METHOD PUBLIC  Clone : I_Node
VAR
	pNode : POINTER TO Node_F_VN_CopyImageRegionToRegion;
END_VAR
pNode := __NEW(Node_F_VN_CopyImageRegionToRegion);
Clone := pNode^;
END_METHOD

METHOD PROTECTED OnExecute
hresult.Value := F_VN_CopyImageRegionToRegion(
    ipSrcImage := ipSrcImage.Value,
    nXSrc := nXSrc.Value,
    nYSrc := nYSrc.Value,
    nWidth := nWidth.Value,
	nHeight := nHeight.Value,
	ipDestImage := ipDestImage.Value,
    nXDest := nXDest.Value,
    nYDest := nYDest.Value,
	hrPrev:= hrPrev.Value);
END_METHOD

METHOD PUBLIC PreExecutionCheck
VAR_INPUT
	Check : I_PreExecutionChecks;
END_VAR
VAR
    imgWidth : UDINT;
    imgHeight : UDINT;
    roiRectangle : TcVnRectangle_UDINT;
END_VAR
Check.IsTrue(ipSrcImage.IsValid, 'ipSrcImage must contain an image');

IF Check.Failed THEN
    RETURN;
END_IF

ipSrcImage.Value.GetWidth(imgWidth);
ipSrcImage.Value.GetHeight(imgHeight);
roiRectangle.nX := nXSrc.Value;
roiRectangle.nY := nYSrc.Value;
roiRectangle.nWidth := nWidth.Value;
roiRectangle.nHeight := nHeight.Value;

Check.IsTrue(IsRoiSizeOK_Udint(roiRectangle, imgWidth, imgHeight), 'ROI must fit within ipSrcImage');

//TODO Check nXDist and nYDest values?
END_METHOD

END_FUNCTION_BLOCK

// Nodes/Basic Image Ops/Node_F_VN_CopyIntoDisplayableImage
{attribute 'linkalways'} 
{attribute 'no_explicit_call' := 'This FB is a CLASS and must be accessed using methods or properties'}
{attribute 'enable_dynamic_creation'}
FUNCTION_BLOCK Node_F_VN_CopyIntoDisplayableImage EXTENDS VisionNode
VAR
    ipSrcImage : _ITcVnImage;
    ipDestImage : _ITcVnDisplayableImage;
    hrPrev : _HRESULT(S_OK);
	hresult : _HRESULT(S_OK);
END_VAR

METHOD FB_init : BOOL
VAR_INPUT
	bInitRetains : BOOL; // if TRUE, the retain variables are initialized (warm start / cold start)
	bInCopyCode : BOOL;  // if TRUE, the instance afterwards gets moved into the copy code (online change)
END_VAR
AddInput('ipSrcImage', ipSrcImage);
AddInput('hrPrev', hrPrev);
AddOutput('ipDestImage', ipDestImage);
AddOutput('hresult',hresult);
END_METHOD

METHOD PUBLIC  Clone : I_Node
VAR
	pNode : POINTER TO Node_F_VN_CopyIntoDisplayableImage;
END_VAR
pNode := __NEW(Node_F_VN_CopyIntoDisplayableImage);
Clone := pNode^;
END_METHOD

METHOD PROTECTED OnExecute
hresult.Value := F_VN_CopyIntoDisplayableImage(
    ipSrcImage := ipSrcImage.Value,
	ipDestImage := ipDestImage.Value,
	hrPrev:= hrPrev.Value);
END_METHOD

METHOD PUBLIC PreExecutionCheck
VAR_INPUT
	Check : I_PreExecutionChecks;
END_VAR
Check.IsTrue(ipSrcImage.IsValid, 'ipSrcImage must contain an image');
END_METHOD

END_FUNCTION_BLOCK

// Nodes/Basic Image Ops/Node_F_VN_CreateAssociatedImage
{attribute 'linkalways'} 
{attribute 'no_explicit_call' := 'This FB is a CLASS and must be accessed using methods or properties'}
{attribute 'enable_dynamic_creation'}
FUNCTION_BLOCK Node_F_VN_CreateAssociatedImage EXTENDS VisionNode
VAR
    ipSrcImage : _ITcVnImage;
    ipDestImage : _ITcVnImage;
    hrPrev : _HRESULT(S_OK);
	hresult : _HRESULT(S_OK);
END_VAR

METHOD FB_init : BOOL
VAR_INPUT
	bInitRetains : BOOL; // if TRUE, the retain variables are initialized (warm start / cold start)
	bInCopyCode : BOOL;  // if TRUE, the instance afterwards gets moved into the copy code (online change)
END_VAR
AddInput('ipSrcImage', ipSrcImage);
AddInput('hrPrev', hrPrev);
AddOutput('ipDestImage', ipDestImage);
AddOutput('hresult',hresult);
END_METHOD

METHOD PUBLIC  Clone : I_Node
VAR
	pNode : POINTER TO Node_F_VN_CreateAssociatedImage;
END_VAR
pNode := __NEW(Node_F_VN_CreateAssociatedImage);
Clone := pNode^;
END_METHOD

METHOD PROTECTED OnExecute
hresult.Value := F_VN_CreateAssociatedImage(
    ipSrcImage := ipSrcImage.Value,
	ipDestImage := ipDestImage.Value,
	hrPrev:= hrPrev.Value);
END_METHOD

METHOD PUBLIC PreExecutionCheck
VAR_INPUT
	Check : I_PreExecutionChecks;
END_VAR
Check.IsTrue(ipSrcImage.IsValid, 'ipSrcImage must contain an image');
END_METHOD

END_FUNCTION_BLOCK

// Nodes/Basic Image Ops/Node_F_VN_CreateEmptyImage
{attribute 'linkalways'} 
{attribute 'no_explicit_call' := 'This FB is a CLASS and must be accessed using methods or properties'}
{attribute 'enable_dynamic_creation'}
FUNCTION_BLOCK Node_F_VN_CreateEmptyImage EXTENDS VisionNode
VAR
    ipImage : _ITcVnImage;
    hrPrev : _HRESULT(S_OK);
	hresult : _HRESULT(S_OK);
END_VAR

METHOD FB_init : BOOL
VAR_INPUT
	bInitRetains : BOOL; // if TRUE, the retain variables are initialized (warm start / cold start)
	bInCopyCode : BOOL;  // if TRUE, the instance afterwards gets moved into the copy code (online change)
END_VAR
AddInput('hrPrev', hrPrev);
AddOutput('ipImage', ipImage);
AddOutput('hresult',hresult);
END_METHOD

METHOD PUBLIC  Clone : I_Node
VAR
	pNode : POINTER TO Node_F_VN_CreateEmptyImage;
END_VAR
pNode := __NEW(Node_F_VN_CreateEmptyImage);
Clone := pNode^;
END_METHOD

METHOD PROTECTED OnExecute
hresult.Value := F_VN_CreateEmptyImage(
    ipImage := ipImage.Value,
	hrPrev:= hrPrev.Value);
END_METHOD

METHOD PUBLIC PreExecutionCheck
VAR_INPUT
	Check : I_PreExecutionChecks;
END_VAR
END_METHOD

END_FUNCTION_BLOCK

// Nodes/Basic Image Ops/Node_F_VN_CreateImage
{attribute 'linkalways'} 
{attribute 'no_explicit_call' := 'This FB is a CLASS and must be accessed using methods or properties'}
{attribute 'enable_dynamic_creation'}
FUNCTION_BLOCK Node_F_VN_CreateImage EXTENDS VisionNode
VAR
    ipImage : _ITcVnImage;
    nWidth : _UDINT(1);
    nHeight : _UDINT(1);
    ePixelType : _ETcVnElementType(ETcVnElementType.TCVN_ET_USINT);
    nChannelNum : _UDINT(1);
    hrPrev : _HRESULT(S_OK);
	hresult : _HRESULT(S_OK);
END_VAR

METHOD FB_init : BOOL
VAR_INPUT
	bInitRetains : BOOL; // if TRUE, the retain variables are initialized (warm start / cold start)
	bInCopyCode : BOOL;  // if TRUE, the instance afterwards gets moved into the copy code (online change)
END_VAR
AddParameter('nWidth', nWidth);
AddParameter('nHeight', nHeight);
AddParameter('ePixelType', ePixelType);
AddParameter('nChannelNum', nChannelNum);
AddInput('hrPrev', hrPrev);
AddOutput('ipImage', ipImage);
AddOutput('hresult',hresult);
END_METHOD

METHOD PUBLIC  Clone : I_Node
VAR
	pNode : POINTER TO Node_F_VN_CreateImage;
END_VAR
pNode := __NEW(Node_F_VN_CreateImage);
Clone := pNode^;
END_METHOD

METHOD PROTECTED OnExecute
hresult.Value := F_VN_CreateImage(
    ipImage := ipImage.Value,
    nWidth := nWidth.Value,
    nHeight := nHeight.Value,
    ePixelType := ePixelType.Value,
    nChannelNum := nChannelNum.Value,
	hrPrev:= hrPrev.Value);
END_METHOD

METHOD PUBLIC PreExecutionCheck
VAR_INPUT
	Check : I_PreExecutionChecks;
END_VAR
Check.IsTrue((nWidth.Value > 0), 'nWidth must be greater than 0');
Check.IsTrue((nHeight.Value > 0), 'nHeight must be greater than 0');
Check.IsTrue((nChannelNum.Value >= 1), 'nChannelNum must be greater than or equal to 1');
Check.IsTrue((nChannelNum.Value <= 255), 'nChannelNum must be less than or equal to 255');
END_METHOD

END_FUNCTION_BLOCK

// Nodes/Basic Image Ops/Node_F_VN_CreateImageAndSetPixels
{attribute 'linkalways'} 
{attribute 'no_explicit_call' := 'This FB is a CLASS and must be accessed using methods or properties'}
{attribute 'enable_dynamic_creation'}
FUNCTION_BLOCK Node_F_VN_CreateImageAndSetPixels EXTENDS VisionNode
VAR
    ipImage : _ITcVnImage;
    nWidth : _UDINT(1);
    nHeight : _UDINT(1);
    ePixelType : _ETcVnElementType(ETcVnElementType.TCVN_ET_USINT);
    nChannelNum : _UDINT(1);
    aValue : _TcVnVector4_LREAL;
    hrPrev : _HRESULT(S_OK);
	hresult : _HRESULT(S_OK);
END_VAR

METHOD FB_init : BOOL
VAR_INPUT
	bInitRetains : BOOL; // if TRUE, the retain variables are initialized (warm start / cold start)
	bInCopyCode : BOOL;  // if TRUE, the instance afterwards gets moved into the copy code (online change)
END_VAR
AddParameter('nWidth', nWidth);
AddParameter('nHeight', nHeight);
AddParameter('ePixelType', ePixelType);
AddParameter('nChannelNum', nChannelNum);
AddInput('aValue', aValue);
AddInput('hrPrev', hrPrev);
AddOutput('ipImage', ipImage);
AddOutput('hresult',hresult);
END_METHOD

METHOD PUBLIC  Clone : I_Node
VAR
	pNode : POINTER TO Node_F_VN_CreateImageAndSetPixels;
END_VAR
pNode := __NEW(Node_F_VN_CreateImageAndSetPixels);
Clone := pNode^;
END_METHOD

METHOD PROTECTED OnExecute
hresult.Value := F_VN_CreateImageAndSetPixels(
    ipImage := ipImage.Value,
    nWidth := nWidth.Value,
    nHeight := nHeight.Value,
    ePixelType := ePixelType.Value,
    nChannelNum := nChannelNum.Value,
    aValue := aValue.Value,
	hrPrev:= hrPrev.Value);
END_METHOD

METHOD PUBLIC PreExecutionCheck
VAR_INPUT
	Check : I_PreExecutionChecks;
END_VAR
Check.IsTrue((nWidth.Value > 0), 'nWidth must be greater than 0');
Check.IsTrue((nHeight.Value > 0), 'nHeight must be greater than 0');
Check.IsTrue((nChannelNum.Value >= 1), 'nChannelNum must be greater than or equal to 1');
Check.IsTrue((nChannelNum.Value <= 4), 'nChannelNum must be less than or equal to 4');
END_METHOD

END_FUNCTION_BLOCK

// Nodes/Basic Image Ops/Node_F_VN_CreateNDimensionalImage
{attribute 'linkalways'} 
{attribute 'no_explicit_call' := 'This FB is a CLASS and must be accessed using methods or properties'}
{attribute 'enable_dynamic_creation'}
FUNCTION_BLOCK Node_F_VN_CreateNDimensionalImage EXTENDS VisionNode
VAR
    ipImage : _ITcVnImage;
    aShape : _TcVnArray33_UDINT;
    ePixelType : _ETcVnElementType(ETcVnElementType.TCVN_ET_USINT);
    hrPrev : _HRESULT(S_OK);
	hresult : _HRESULT(S_OK);
END_VAR

METHOD FB_init : BOOL
VAR_INPUT
	bInitRetains : BOOL; // if TRUE, the retain variables are initialized (warm start / cold start)
	bInCopyCode : BOOL;  // if TRUE, the instance afterwards gets moved into the copy code (online change)
END_VAR
AddParameter('aShape', aShape);
AddParameter('ePixelType', ePixelType);
AddInput('hrPrev', hrPrev);
AddOutput('ipImage', ipImage);
AddOutput('hresult',hresult);
END_METHOD

METHOD PUBLIC  Clone : I_Node
VAR
	pNode : POINTER TO Node_F_VN_CreateNDimensionalImage;
END_VAR
pNode := __NEW(Node_F_VN_CreateNDimensionalImage);
Clone := pNode^;
END_METHOD

METHOD PROTECTED OnExecute
hresult.Value := F_VN_CreateNDimensionalImage(
    ipImage := ipImage.Value,
    aShape := aShape.Value,
    ePixelType := ePixelType.Value,
	hrPrev:= hrPrev.Value);
END_METHOD

METHOD PUBLIC PreExecutionCheck
VAR_INPUT
	Check : I_PreExecutionChecks;
END_VAR
END_METHOD

END_FUNCTION_BLOCK

// Nodes/Basic Image Ops/Node_F_VN_CreateNDimensionalImageAndSetPixels
{attribute 'linkalways'} 
{attribute 'no_explicit_call' := 'This FB is a CLASS and must be accessed using methods or properties'}
{attribute 'enable_dynamic_creation'}
FUNCTION_BLOCK Node_F_VN_CreateNDimensionalImageAndSetPixels EXTENDS VisionNode
VAR
    ipImage : _ITcVnImage;
    aShape : _TcVnArray33_UDINT;
    ePixelType : _ETcVnElementType(ETcVnElementType.TCVN_ET_USINT);
    fValue : _LREAL(0.0);
    hrPrev : _HRESULT(S_OK);
	hresult : _HRESULT(S_OK);
END_VAR

METHOD FB_init : BOOL
VAR_INPUT
	bInitRetains : BOOL; // if TRUE, the retain variables are initialized (warm start / cold start)
	bInCopyCode : BOOL;  // if TRUE, the instance afterwards gets moved into the copy code (online change)
END_VAR
AddParameter('aShape', aShape);
AddParameter('ePixelType', ePixelType);
AddParameter('fValue', fValue);
AddInput('hrPrev', hrPrev);
AddOutput('ipImage', ipImage);
AddOutput('hresult',hresult);
END_METHOD

METHOD PUBLIC  Clone : I_Node
VAR
	pNode : POINTER TO Node_F_VN_CreateNDimensionalImageAndSetPixels;
END_VAR
pNode := __NEW(Node_F_VN_CreateNDimensionalImageAndSetPixels);
Clone := pNode^;
END_METHOD

METHOD PROTECTED OnExecute
hresult.Value := F_VN_CreateNDimensionalImageAndSetPixels(
    ipImage := ipImage.Value,
    aShape := aShape.Value,
    ePixelType := ePixelType.Value,
    fValue := fValue.Value,
	hrPrev:= hrPrev.Value);
END_METHOD

METHOD PUBLIC PreExecutionCheck
VAR_INPUT
	Check : I_PreExecutionChecks;
END_VAR
END_METHOD

END_FUNCTION_BLOCK

// Nodes/Basic Image Ops/Node_F_VN_ExportImageAsBmpSize
{attribute 'linkalways'} 
{attribute 'no_explicit_call' := 'This FB is a CLASS and must be accessed using methods or properties'}
{attribute 'enable_dynamic_creation'}
FUNCTION_BLOCK Node_F_VN_ExportImageAsBmpSize EXTENDS VisionNode
VAR
    ipImage : _ITcVnImage;
    nBufferSize : _ULINT(0);
    hrPrev : _HRESULT(S_OK);
	hresult : _HRESULT(S_OK);
END_VAR

METHOD FB_init : BOOL
VAR_INPUT
	bInitRetains : BOOL; // if TRUE, the retain variables are initialized (warm start / cold start)
	bInCopyCode : BOOL;  // if TRUE, the instance afterwards gets moved into the copy code (online change)
END_VAR
AddInput('ipImage', ipImage);
AddInput('hrPrev', hrPrev);
AddOutput('nBufferSize', nBufferSize);
AddOutput('hresult',hresult);
END_METHOD

METHOD PUBLIC  Clone : I_Node
VAR
	pNode : POINTER TO Node_F_VN_ExportImageAsBmpSize;
END_VAR
pNode := __NEW(Node_F_VN_ExportImageAsBmpSize);
Clone := pNode^;
END_METHOD

METHOD PROTECTED OnExecute
hresult.Value := F_VN_ExportImageAsBmpSize(
    ipImage := ipImage.Value,
    nBufferSize := nBufferSize.Value,
	hrPrev:= hrPrev.Value);
END_METHOD

METHOD PUBLIC PreExecutionCheck
VAR_INPUT
	Check : I_PreExecutionChecks;
END_VAR
Check.IsTrue(ipImage.IsValid, 'ipImage must contain an image');
END_METHOD

END_FUNCTION_BLOCK

// Nodes/Basic Image Ops/Node_F_VN_ExportImageAsBmpSizeExp
{attribute 'linkalways'} 
{attribute 'no_explicit_call' := 'This FB is a CLASS and must be accessed using methods or properties'}
{attribute 'enable_dynamic_creation'}
FUNCTION_BLOCK Node_F_VN_ExportImageAsBmpSizeExp EXTENDS VisionNode
VAR
    ipImage : _ITcVnImage;
    nBufferSize : _ULINT(0);
    nWidth : _UDINT(0);
    nHeight : _UDINT(0);
    hrPrev : _HRESULT(S_OK);
	hresult : _HRESULT(S_OK);
END_VAR

METHOD FB_init : BOOL
VAR_INPUT
	bInitRetains : BOOL; // if TRUE, the retain variables are initialized (warm start / cold start)
	bInCopyCode : BOOL;  // if TRUE, the instance afterwards gets moved into the copy code (online change)
END_VAR
AddInput('ipImage', ipImage);
AddParameter('nWidth', nWidth);
AddParameter('nHeight', nHeight);
AddInput('hrPrev', hrPrev);
AddOutput('nBufferSize', nBufferSize);
AddOutput('hresult', hresult);
END_METHOD

METHOD PUBLIC  Clone : I_Node
VAR
	pNode : POINTER TO Node_F_VN_ExportImageAsBmpSizeExp;
END_VAR
pNode := __NEW(Node_F_VN_ExportImageAsBmpSizeExp);
Clone := pNode^;
END_METHOD

METHOD PROTECTED OnExecute
hresult.Value := F_VN_ExportImageAsBmpSizeExp(
    ipImage := ipImage.Value,
    nBufferSize := nBufferSize.Value,
    nWidth := nWidth.Value,
    nHeight := nHeight.Value,
	hrPrev:= hrPrev.Value);
END_METHOD

METHOD PUBLIC PreExecutionCheck
VAR_INPUT
	Check : I_PreExecutionChecks;
END_VAR
Check.IsTrue(ipImage.IsValid, 'ipImage must contain an image');
END_METHOD

END_FUNCTION_BLOCK

// Nodes/Basic Image Ops/Node_F_VN_ExportImageSize
{attribute 'linkalways'} 
{attribute 'no_explicit_call' := 'This FB is a CLASS and must be accessed using methods or properties'}
{attribute 'enable_dynamic_creation'}
FUNCTION_BLOCK Node_F_VN_ExportImageSize EXTENDS VisionNode
VAR
    ipImage : _ITcVnImage;
    nBufferSize : _ULINT(0);
    hrPrev : _HRESULT(S_OK);
	hresult : _HRESULT(S_OK);
END_VAR

METHOD FB_init : BOOL
VAR_INPUT
	bInitRetains : BOOL; // if TRUE, the retain variables are initialized (warm start / cold start)
	bInCopyCode : BOOL;  // if TRUE, the instance afterwards gets moved into the copy code (online change)
END_VAR
AddInput('ipImage', ipImage);
AddInput('hrPrev', hrPrev);
AddOutput('nBufferSize', nBufferSize);
AddOutput('hresult',hresult);
END_METHOD

METHOD PUBLIC  Clone : I_Node
VAR
	pNode : POINTER TO Node_F_VN_ExportImageSize;
END_VAR
pNode := __NEW(Node_F_VN_ExportImageSize);
Clone := pNode^;
END_METHOD

METHOD PROTECTED OnExecute
hresult.Value := F_VN_ExportImageSize(
    ipImage := ipImage.Value,
    nBufferSize := nBufferSize.Value,
	hrPrev:= hrPrev.Value);
END_METHOD

METHOD PUBLIC PreExecutionCheck
VAR_INPUT
	Check : I_PreExecutionChecks;
END_VAR
Check.IsTrue(ipImage.IsValid, 'ipImage must contain an image');
END_METHOD

END_FUNCTION_BLOCK

// Nodes/Basic Image Ops/Node_F_VN_FuseImages
{attribute 'linkalways'} 
{attribute 'no_explicit_call' := 'This FB is a CLASS and must be accessed using methods or properties'}
{attribute 'enable_dynamic_creation'}
FUNCTION_BLOCK Node_F_VN_FuseImages EXTENDS VisionNode
VAR
    ipSrcImage1 : _ITcVnImage;
    ipSrcImage2 : _ITcVnImage;
    ipDestImage : _ITcVnImage;
    nFirstLine : _UDINT(0);
    nNumLines : _UDINT(0);
    hrPrev : _HRESULT(S_OK);
	hresult : _HRESULT(S_OK);
END_VAR

METHOD FB_init : BOOL
VAR_INPUT
	bInitRetains : BOOL; // if TRUE, the retain variables are initialized (warm start / cold start)
	bInCopyCode : BOOL;  // if TRUE, the instance afterwards gets moved into the copy code (online change)
END_VAR
AddInput('ipSrcImage1', ipSrcImage1);
AddInput('ipSrcImage2', ipSrcImage2);
AddParameter('nFirstLine', nFirstLine);
AddParameter('nNumLines', nNumLines);
AddInput('hrPrev', hrPrev);
AddOutput('ipDestImage', ipDestImage);
AddOutput('hresult',hresult);
END_METHOD

METHOD PUBLIC  Clone : I_Node
VAR
	pNode : POINTER TO Node_F_VN_FuseImages;
END_VAR
pNode := __NEW(Node_F_VN_FuseImages);
Clone := pNode^;
END_METHOD

METHOD PROTECTED OnExecute
hresult.Value := F_VN_FuseImages(
    ipSrcImage1 := ipSrcImage1.Value,
    ipSrcImage2 := ipSrcImage2.Value,
	ipDestImage := ipDestImage.Value,
    nFirstLine := nFirstLine.Value,
    nNumLines := nNumLines.Value,
	hrPrev:= hrPrev.Value);
END_METHOD

METHOD PUBLIC PreExecutionCheck
VAR_INPUT
	Check : I_PreExecutionChecks;
END_VAR
Check.IsTrue(ipSrcImage1.IsValid, 'ipSrcImage1 must contain an image');
Check.IsTrue(ipSrcImage2.IsValid, 'ipSrcImage2 must contain an image');
Check.IsTrue(IsImage1WidthEqualToImage2Width(ipSrcImage1.Value, ipSrcImage2.Value), 'ipSrcImage1 must be the same width as ipSrcImage2');
Check.IsTrue(ImagesHaveMatchingPixelFormats(ipSrcImage1.Value, ipSrcImage2.Value), 'ipSrcImage2 must have same pixel depth as ipSrcImage1');
END_METHOD

END_FUNCTION_BLOCK

// Nodes/Basic Image Ops/Node_F_VN_GetImageChannel
{attribute 'linkalways'} 
{attribute 'no_explicit_call' := 'This FB is a CLASS and must be accessed using methods or properties'}
{attribute 'enable_dynamic_creation'}
FUNCTION_BLOCK Node_F_VN_GetImageChannel EXTENDS VisionNode
VAR
    ipSrcImage : _ITcVnImage;
    ipDestImage : _ITcVnImage;
    nChannelIndex : _UINT(0);
    hrPrev : _HRESULT(S_OK);
	hresult : _HRESULT(S_OK);
END_VAR

METHOD FB_init : BOOL
VAR_INPUT
	bInitRetains : BOOL; // if TRUE, the retain variables are initialized (warm start / cold start)
	bInCopyCode : BOOL;  // if TRUE, the instance afterwards gets moved into the copy code (online change)
END_VAR
AddInput('ipSrcImage', ipSrcImage);
AddInput('hrPrev', hrPrev);
AddOutput('ipDestImage', ipDestImage);
AddOutput('hresult',hresult);
AddParameter('nChannelIndex', nChannelIndex);
END_METHOD

METHOD PUBLIC  Clone : I_Node
VAR
	pNode : POINTER TO Node_F_VN_GetImageChannel;
END_VAR
pNode := __NEW(Node_F_VN_GetImageChannel);
Clone := pNode^;
END_METHOD

METHOD PROTECTED OnExecute
// ----------------------------------------------------------------------------
// TcVision 4.0.6.5, 4.0.7.4 BUG FIX
// ----------------------------------------------------------------------------
// Get Image Channel fails, if used on two different sized images, 
// without clearing the destination image first. 
// so, we check to see if hrPrev is failed, in which case we do nothing
// as the function would do nothing natively.  Else, we check the dest
// image, and if it has something, it is first emptied
// ---------------------------------------------------------------------------- 
IF failed(hrPrev.Value) THEN
	RETURN;
END_IF

IF ipDestImage.IsValid THEN
	ipDestImage.Value.TcRelease();
	ipDestImage.Value := 0;
END_IF
// ---------------------------------------------------------------------------- 

hresult.Value := F_VN_GetImageChannel(
    ipSrcImage := ipSrcImage.Value,
	ipDestImage := ipDestImage.Value,
    nChannelIndex := nChannelIndex.Value,
	hrPrev:= hrPrev.Value);
END_METHOD

METHOD PUBLIC PreExecutionCheck
VAR_INPUT
	Check : I_PreExecutionChecks;
END_VAR
Check.IsTrue(ipSrcImage.IsValid, 'ipSrcImage must contain an image');
END_METHOD

END_FUNCTION_BLOCK

// Nodes/Basic Image Ops/Node_F_VN_GetImageHeight
{attribute 'linkalways'} 
{attribute 'no_explicit_call' := 'This FB is a CLASS and must be accessed using methods or properties'}
{attribute 'enable_dynamic_creation'}
FUNCTION_BLOCK Node_F_VN_GetImageHeight EXTENDS VisionNode
VAR
    ipImage : _ITcVnImage;
    nHeight : _UDINT(0);
    hrPrev : _HRESULT(S_OK);
	hresult : _HRESULT(S_OK);
END_VAR

METHOD FB_init : BOOL
VAR_INPUT
	bInitRetains : BOOL; // if TRUE, the retain variables are initialized (warm start / cold start)
	bInCopyCode : BOOL;  // if TRUE, the instance afterwards gets moved into the copy code (online change)
END_VAR
AddInput('ipImage', ipImage);
AddInput('hrPrev', hrPrev);
AddOutput('nHeight', nHeight);
AddOutput('hresult', hresult);
END_METHOD

METHOD PUBLIC  Clone : I_Node
VAR
	pNode : POINTER TO Node_F_VN_GetImageHeight;
END_VAR
pNode := __NEW(Node_F_VN_GetImageHeight);
Clone := pNode^;
END_METHOD

METHOD PROTECTED OnExecute
hresult.Value := F_VN_GetImageHeight(
    ipImage := ipImage.Value,
    nHeight := nHeight.Value,
	hrPrev:= hrPrev.Value);
END_METHOD

METHOD PUBLIC PreExecutionCheck
VAR_INPUT
	Check : I_PreExecutionChecks;
END_VAR
Check.IsTrue(ipImage.IsValid, 'ipImage must contain an image');
END_METHOD

END_FUNCTION_BLOCK

// Nodes/Basic Image Ops/Node_F_VN_GetImageInfo
{attribute 'linkalways'} 
{attribute 'no_explicit_call' := 'This FB is a CLASS and must be accessed using methods or properties'}
{attribute 'enable_dynamic_creation'}
FUNCTION_BLOCK Node_F_VN_GetImageInfo EXTENDS VisionNode
VAR
    ipImage : _ITcVnImage;
    stImageInfo : _TcVnImageInfo;
    hrPrev : _HRESULT(S_OK);
	hresult : _HRESULT(S_OK);
END_VAR

METHOD FB_init : BOOL
VAR_INPUT
	bInitRetains : BOOL; // if TRUE, the retain variables are initialized (warm start / cold start)
	bInCopyCode : BOOL;  // if TRUE, the instance afterwards gets moved into the copy code (online change)
END_VAR
AddInput('ipImage', ipImage);
AddInput('hrPrev', hrPrev);
AddOutput('stImageInfo', stImageInfo);
AddOutput('hresult',hresult);
END_METHOD

METHOD PUBLIC  Clone : I_Node
VAR
	pNode : POINTER TO Node_F_VN_GetImageInfo;
END_VAR
pNode := __NEW(Node_F_VN_GetImageInfo);
Clone := pNode^;
END_METHOD

METHOD PROTECTED OnExecute
hresult.Value := F_VN_GetImageInfo(
    ipImage := ipImage.Value,
	stImageInfo := stImageInfo.Value,
	hrPrev:= hrPrev.Value);
END_METHOD

METHOD PUBLIC PreExecutionCheck
VAR_INPUT
	Check : I_PreExecutionChecks;
END_VAR
Check.IsTrue(ipImage.IsValid, 'ipImage must contain an image');
END_METHOD

END_FUNCTION_BLOCK

// Nodes/Basic Image Ops/Node_F_VN_GetImageWidth
{attribute 'linkalways'} 
{attribute 'no_explicit_call' := 'This FB is a CLASS and must be accessed using methods or properties'}
{attribute 'enable_dynamic_creation'}
FUNCTION_BLOCK Node_F_VN_GetImageWidth EXTENDS VisionNode
VAR
    ipImage : _ITcVnImage;
    nWidth : _UDINT(0);
    hrPrev : _HRESULT(S_OK);
	hresult : _HRESULT(S_OK);
END_VAR

METHOD FB_init : BOOL
VAR_INPUT
	bInitRetains : BOOL; // if TRUE, the retain variables are initialized (warm start / cold start)
	bInCopyCode : BOOL;  // if TRUE, the instance afterwards gets moved into the copy code (online change)
END_VAR
AddInput('ipImage', ipImage);
AddInput('hrPrev', hrPrev);
AddOutput('nWidth', nWidth);
AddOutput('hresult',hresult);
END_METHOD

METHOD PUBLIC  Clone : I_Node
VAR
	pNode : POINTER TO Node_F_VN_GetImageWidth;
END_VAR
pNode := __NEW(Node_F_VN_GetImageWidth);
Clone := pNode^;
END_METHOD

METHOD PROTECTED OnExecute
hresult.Value := F_VN_GetImageWidth(
    ipImage := ipImage.Value,
    nWidth := nWidth.Value,
	hrPrev:= hrPrev.Value);
END_METHOD

METHOD PUBLIC PreExecutionCheck
VAR_INPUT
	Check : I_PreExecutionChecks;
END_VAR
Check.IsTrue(ipImage.IsValid, 'ipImage must contain an image');
END_METHOD

END_FUNCTION_BLOCK

// Nodes/Basic Image Ops/Node_F_VN_GetLayoutInfo
{attribute 'linkalways'} 
{attribute 'no_explicit_call' := 'This FB is a CLASS and must be accessed using methods or properties'}
{attribute 'enable_dynamic_creation'}
FUNCTION_BLOCK Node_F_VN_GetLayoutInfo EXTENDS VisionNode
VAR
    ipImage : _ITcVnImage;
    aLayoutInfo : _TcVnArray33_UDINT;
    hrPrev : _HRESULT(S_OK);
	hresult : _HRESULT(S_OK);
END_VAR

METHOD FB_init : BOOL
VAR_INPUT
	bInitRetains : BOOL; // if TRUE, the retain variables are initialized (warm start / cold start)
	bInCopyCode : BOOL;  // if TRUE, the instance afterwards gets moved into the copy code (online change)
END_VAR
AddInput('ipImage', ipImage);
AddInput('hrPrev', hrPrev);
AddOutput('aLayoutInfo', aLayoutInfo);
AddOutput('hresult',hresult);
END_METHOD

METHOD PUBLIC  Clone : I_Node
VAR
	pNode : POINTER TO Node_F_VN_GetLayoutInfo;
END_VAR
pNode := __NEW(Node_F_VN_GetLayoutInfo);
Clone := pNode^;
END_METHOD

METHOD PROTECTED OnExecute
hresult.Value := F_VN_GetLayoutInfo(
    ipImage := ipImage.Value,
	aLayoutInfo := aLayoutInfo.Value,
	hrPrev:= hrPrev.Value);
END_METHOD

METHOD PUBLIC PreExecutionCheck
VAR_INPUT
	Check : I_PreExecutionChecks;
END_VAR
Check.IsTrue(ipImage.IsValid, 'ipImage must contain an image');
END_METHOD

END_FUNCTION_BLOCK

// Nodes/Basic Image Ops/Node_F_VN_GetPixel
{attribute 'linkalways'} 
{attribute 'no_explicit_call' := 'This FB is a CLASS and must be accessed using methods or properties'}
{attribute 'enable_dynamic_creation'}
FUNCTION_BLOCK Node_F_VN_GetPixel EXTENDS VisionNode
VAR
    ipSrcImage : _ITcVnImage;
    aValue : _TcVnVector4_LREAL;
    nX : _UDINT(0);
    nY : _UDINT(0);
    hrPrev : _HRESULT(S_OK);
	hresult : _HRESULT(S_OK);
END_VAR

METHOD FB_init : BOOL
VAR_INPUT
	bInitRetains : BOOL; // if TRUE, the retain variables are initialized (warm start / cold start)
	bInCopyCode : BOOL;  // if TRUE, the instance afterwards gets moved into the copy code (online change)
END_VAR
AddInput('ipSrcImage', ipSrcImage);
AddParameter('nX', nX);
AddParameter('nY', nY);
AddInput('hrPrev', hrPrev);
AddOutput('aValue', aValue);
AddOutput('hresult',hresult);
END_METHOD

METHOD PUBLIC  Clone : I_Node
VAR
	pNode : POINTER TO Node_F_VN_GetPixel;
END_VAR
pNode := __NEW(Node_F_VN_GetPixel);
Clone := pNode^;
END_METHOD

METHOD PROTECTED OnExecute
hresult.Value := F_VN_GetPixel(
    ipSrcImage := ipSrcImage.Value,
    aValue := aValue.Value,
    nX := nX.Value,
    nY := nY.Value,
	hrPrev:= hrPrev.Value);
END_METHOD

METHOD PUBLIC PreExecutionCheck
VAR_INPUT
	Check : I_PreExecutionChecks;
END_VAR
Check.IsTrue(ipSrcImage.IsValid, 'ipSrcImage must contain an image');
END_METHOD

END_FUNCTION_BLOCK

// Nodes/Basic Image Ops/Node_F_VN_GetPixelFormat
{attribute 'linkalways'} 
{attribute 'no_explicit_call' := 'This FB is a CLASS and must be accessed using methods or properties'}
{attribute 'enable_dynamic_creation'}
FUNCTION_BLOCK Node_F_VN_GetPixelFormat EXTENDS VisionNode
VAR
    ipImage : _ITcVnImage;
    stPixelFormat : _TcVnPixelFormat;
    hrPrev : _HRESULT(S_OK);
	hresult : _HRESULT(S_OK);
END_VAR

METHOD FB_init : BOOL
VAR_INPUT
	bInitRetains : BOOL; // if TRUE, the retain variables are initialized (warm start / cold start)
	bInCopyCode : BOOL;  // if TRUE, the instance afterwards gets moved into the copy code (online change)
END_VAR
AddInput('ipImage', ipImage);
AddInput('hrPrev', hrPrev);
AddOutput('stPixelFormat', stPixelFormat);
AddOutput('hresult',hresult);
END_METHOD

METHOD PUBLIC  Clone : I_Node
VAR
	pNode : POINTER TO Node_F_VN_GetPixelFormat;
END_VAR
pNode := __NEW(Node_F_VN_GetPixelFormat);
Clone := pNode^;
END_METHOD

METHOD PROTECTED OnExecute
hresult.Value := F_VN_GetPixelFormat(
    ipImage := ipImage.Value,
	stPixelFormat := stPixelFormat.Value,
	hrPrev:= hrPrev.Value);
END_METHOD

METHOD PUBLIC PreExecutionCheck
VAR_INPUT
	Check : I_PreExecutionChecks;
END_VAR
Check.IsTrue(ipImage.IsValid, 'ipImage must contain an image');
END_METHOD

END_FUNCTION_BLOCK

// Nodes/Basic Image Ops/Node_F_VN_GetRoi
{attribute 'linkalways'} 
{attribute 'no_explicit_call' := 'This FB is a CLASS and must be accessed using methods or properties'}
{attribute 'enable_dynamic_creation'}
FUNCTION_BLOCK Node_F_VN_GetRoi EXTENDS VisionNode
VAR
    ipSrcImage : _ITcVnImage;
    stRoi : _TcVnRectangle_UDINT;
    hrPrev : _HRESULT(S_OK);
	hresult : _HRESULT(S_OK);
END_VAR

METHOD FB_init : BOOL
VAR_INPUT
	bInitRetains : BOOL; // if TRUE, the retain variables are initialized (warm start / cold start)
	bInCopyCode : BOOL;  // if TRUE, the instance afterwards gets moved into the copy code (online change)
END_VAR
AddInput('ipSrcImage', ipSrcImage);
AddInput('hrPrev', hrPrev);
AddOutput('stRoi', stRoi);
AddOutput('hresult',hresult);
END_METHOD

METHOD PUBLIC  Clone : I_Node
VAR
	pNode : POINTER TO Node_F_VN_GetRoi;
END_VAR
pNode := __NEW(Node_F_VN_GetRoi);
Clone := pNode^;
END_METHOD

METHOD PROTECTED OnExecute
hresult.Value := F_VN_GetRoi(
    ipSrcImage := ipSrcImage.Value,
    stRoi := stRoi.Value,
	hrPrev:= hrPrev.Value);
END_METHOD

METHOD PUBLIC PreExecutionCheck
VAR_INPUT
	Check : I_PreExecutionChecks;
END_VAR
Check.IsTrue(ipSrcImage.IsValid, 'ipSrcImage must contain an image');
END_METHOD

END_FUNCTION_BLOCK

// Nodes/Basic Image Ops/Node_F_VN_MixImageChannels
{attribute 'linkalways'} 
{attribute 'no_explicit_call' := 'This FB is a CLASS and must be accessed using methods or properties'}
{attribute 'enable_dynamic_creation'}
FUNCTION_BLOCK Node_F_VN_MixImageChannels EXTENDS VisionNode
VAR
    ipSrcImage : _ITcVnImage;
    ipDestImage : _ITcVnImage;
    ipIndicesFromTo : _ITcVnContainer;
    hrPrev : _HRESULT(S_OK);
	hresult : _HRESULT(S_OK);
END_VAR

METHOD FB_init : BOOL
VAR_INPUT
	bInitRetains : BOOL; // if TRUE, the retain variables are initialized (warm start / cold start)
	bInCopyCode : BOOL;  // if TRUE, the instance afterwards gets moved into the copy code (online change)
END_VAR
AddInput('ipSrcImage', ipSrcImage);
AddInput('ipIndicesFromTo', ipIndicesFromTo);
AddInput('hrPrev', hrPrev);
AddOutput('ipDestImage', ipDestImage);
AddOutput('hresult',hresult);
END_METHOD

METHOD PUBLIC  Clone : I_Node
VAR
	pNode : POINTER TO Node_F_VN_MixImageChannels;
END_VAR
pNode := __NEW(Node_F_VN_MixImageChannels);
Clone := pNode^;
END_METHOD

METHOD PROTECTED OnExecute
hresult.Value := F_VN_MixImageChannels(
    ipSrcImage := ipSrcImage.Value,
	ipDestImage := ipDestImage.Value,
    ipIndicesFromTo := ipIndicesFromTo.Value,
	hrPrev := hrPrev.Value);
END_METHOD

METHOD PUBLIC PreExecutionCheck
VAR_INPUT
	Check : I_PreExecutionChecks;
END_VAR
Check.IsTrue(ipSrcImage.IsValid, 'ipSrcImage must contain an image');
Check.IsTrue(ipIndicesFromTo.IsType(TC_GLOBAL_CONST_LIST.ContainerType_Vector_TcVnVector2_DINT),
              'ipIndicesFromTo contains incorrect type');
END_METHOD

END_FUNCTION_BLOCK

// Nodes/Basic Image Ops/Node_F_VN_PadImageBorder
{attribute 'linkalways'} 
{attribute 'no_explicit_call' := 'This FB is a CLASS and must be accessed using methods or properties'}
{attribute 'enable_dynamic_creation'}
FUNCTION_BLOCK Node_F_VN_PadImageBorder EXTENDS VisionNode
VAR
    ipSrcImage : _ITcVnImage;
    ipPaddedImage : _ITcVnImage;
    nTopBorder : _UDINT(0);
    nBottomBorder : _UDINT(0);
    nLeftBorder : _UDINT(0);
    nRightBorder : _UDINT(0);
    hrPrev : _HRESULT(S_OK);
	hresult : _HRESULT(S_OK);
END_VAR

METHOD FB_init : BOOL
VAR_INPUT
	bInitRetains : BOOL; // if TRUE, the retain variables are initialized (warm start / cold start)
	bInCopyCode : BOOL;  // if TRUE, the instance afterwards gets moved into the copy code (online change)
END_VAR
AddInput('ipSrcImage', ipSrcImage);
AddParameter('nTopBorder', nTopBorder);
AddParameter('nBottomBorder', nBottomBorder);
AddParameter('nLeftBorder', nLeftBorder);
AddParameter('nRightBorder', nRightBorder);
AddInput('hrPrev', hrPrev);
AddOutput('ipPaddedImage', ipPaddedImage);
AddOutput('hresult',hresult);
END_METHOD

METHOD PUBLIC  Clone : I_Node
VAR
	pNode : POINTER TO Node_F_VN_PadImageBorder;
END_VAR
pNode := __NEW(Node_F_VN_PadImageBorder);
Clone := pNode^;
END_METHOD

METHOD PROTECTED OnExecute
hresult.Value := F_VN_PadImageBorder(
    ipSrcImage := ipSrcImage.Value,
	ipPaddedImage := ipPaddedImage.Value,
    nTopBorder := nTopBorder.Value,
    nBottomBorder := nBottomBorder.Value,
    nLeftBorder := nLeftBorder.Value,
    nRightBorder := nRightBorder.Value,
	hrPrev:= hrPrev.Value);
END_METHOD

METHOD PUBLIC PreExecutionCheck
VAR_INPUT
	Check : I_PreExecutionChecks;
END_VAR
Check.IsTrue(ipSrcImage.IsValid, 'ipSrcImage must contain an image');
END_METHOD

END_FUNCTION_BLOCK

// Nodes/Basic Image Ops/Node_F_VN_PadImageBorderExp
{attribute 'linkalways'} 
{attribute 'no_explicit_call' := 'This FB is a CLASS and must be accessed using methods or properties'}
{attribute 'enable_dynamic_creation'}
FUNCTION_BLOCK Node_F_VN_PadImageBorderExp EXTENDS VisionNode
VAR
    ipSrcImage : _ITcVnImage;
    ipPaddedImage : _ITcVnImage;
    nTopBorder : _UDINT(0);
    nBottomBorder : _UDINT(0);
    nLeftBorder : _UDINT(0);
    nRightBorder : _UDINT(0);
    ePaddingType : _ETcVnBorderInterpolationMethod(ETcVnBorderInterpolationMethod.TCVN_BIM_CONSTANT);
    aPaddingValue : _TcVnVector4_LREAL;
    hrPrev : _HRESULT(S_OK);
	hresult : _HRESULT(S_OK);
END_VAR

METHOD FB_init : BOOL
VAR_INPUT
	bInitRetains : BOOL; // if TRUE, the retain variables are initialized (warm start / cold start)
	bInCopyCode : BOOL;  // if TRUE, the instance afterwards gets moved into the copy code (online change)
END_VAR
AddInput('ipSrcImage', ipSrcImage);
AddParameter('nTopBorder', nTopBorder);
AddParameter('nBottomBorder', nBottomBorder);
AddParameter('nLeftBorder', nLeftBorder);
AddParameter('nRightBorder', nRightBorder);
AddParameter('ePaddingType', ePaddingType);
AddInput('aPaddingValue', aPaddingValue);
AddInput('hrPrev', hrPrev);
AddOutput('ipPaddedImage', ipPaddedImage);
AddOutput('hresult',hresult);
END_METHOD

METHOD PUBLIC  Clone : I_Node
VAR
	pNode : POINTER TO Node_F_VN_PadImageBorderExp;
END_VAR
pNode := __NEW(Node_F_VN_PadImageBorderExp);
Clone := pNode^;
END_METHOD

METHOD PROTECTED OnExecute
hresult.Value := F_VN_PadImageBorderExp(
    ipSrcImage := ipSrcImage.Value,
	ipPaddedImage := ipPaddedImage.Value,
    nTopBorder := nTopBorder.Value,
    nBottomBorder := nBottomBorder.Value,
    nLeftBorder := nLeftBorder.Value,
    nRightBorder := nRightBorder.Value,
    ePaddingType := ePaddingType.Value,
    aPaddingValue := aPaddingValue.Value,
	hrPrev:= hrPrev.Value);
END_METHOD

METHOD PUBLIC PreExecutionCheck
VAR_INPUT
	Check : I_PreExecutionChecks;
END_VAR
Check.IsTrue(ipSrcImage.IsValid, 'ipSrcImage must contain an image');
END_METHOD

END_FUNCTION_BLOCK

// Nodes/Basic Image Ops/Node_F_VN_ResetRoi
{attribute 'linkalways'} 
{attribute 'no_explicit_call' := 'This FB is a CLASS and must be accessed using methods or properties'}
{attribute 'enable_dynamic_creation'}
FUNCTION_BLOCK Node_F_VN_ResetRoi EXTENDS VisionNode
VAR
    ipImage : _ITcVnImage;
    hrPrev : _HRESULT(S_OK);
	hresult : _HRESULT(S_OK);
END_VAR

METHOD FB_init : BOOL
VAR_INPUT
	bInitRetains : BOOL; // if TRUE, the retain variables are initialized (warm start / cold start)
	bInCopyCode : BOOL;  // if TRUE, the instance afterwards gets moved into the copy code (online change)
END_VAR
AddInput('ipImage', ipImage);
AddInput('hrPrev', hrPrev);
AddOutput('ipImage', ipImage);
AddOutput('hresult', hresult);
END_METHOD

METHOD PUBLIC  Clone : I_Node
VAR
	pNode : POINTER TO Node_F_VN_ResetRoi;
END_VAR
pNode := __NEW(Node_F_VN_ResetRoi);
Clone := pNode^;
END_METHOD

METHOD PROTECTED OnExecute
hresult.Value := F_VN_ResetRoi(
    ipImage := ipImage.Value,
	hrPrev:= hrPrev.Value);
END_METHOD

METHOD PUBLIC PreExecutionCheck
VAR_INPUT
	Check : I_PreExecutionChecks;
END_VAR
Check.IsTrue(ipImage.IsValid, 'ipImage must contain an image');
END_METHOD

END_FUNCTION_BLOCK

// Nodes/Basic Image Ops/Node_F_VN_SetImageChannel
{attribute 'linkalways'} 
{attribute 'no_explicit_call' := 'This FB is a CLASS and must be accessed using methods or properties'}
{attribute 'enable_dynamic_creation'}
FUNCTION_BLOCK Node_F_VN_SetImageChannel EXTENDS VisionNode
VAR
    ipSrcImage : _ITcVnImage;
    ipDestImage : _ITcVnImage;
    nSrcChannelIndex : _UINT(0);
    nDestChannelIndex : _UINT(0);
    hrPrev : _HRESULT(S_OK);
	hresult : _HRESULT(S_OK);
END_VAR

METHOD FB_init : BOOL
VAR_INPUT
	bInitRetains : BOOL; // if TRUE, the retain variables are initialized (warm start / cold start)
	bInCopyCode : BOOL;  // if TRUE, the instance afterwards gets moved into the copy code (online change)
END_VAR
AddInput('ipSrcImage', ipSrcImage);
AddInput('ipDestImage', ipDestImage);
AddParameter('nSrcChannelIndex', nSrcChannelIndex);
AddParameter('nDestChannelIndex', nDestChannelIndex);
AddInput('hrPrev', hrPrev);
AddOutput('ipDestImage', ipDestImage);
AddOutput('hresult',hresult);
END_METHOD

METHOD PUBLIC  Clone : I_Node
VAR
	pNode : POINTER TO Node_F_VN_SetImageChannel;
END_VAR
pNode := __NEW(Node_F_VN_SetImageChannel);
Clone := pNode^;
END_METHOD

METHOD PROTECTED OnExecute
hresult.Value := F_VN_SetImageChannel(
    ipSrcImage := ipSrcImage.Value,
	ipDestImage := ipDestImage.Value,
    nSrcChannelIndex := nSrcChannelIndex.Value,
    nDestChannelIndex := nDestChannelIndex.Value,
	hrPrev:= hrPrev.Value);
END_METHOD

METHOD PUBLIC PreExecutionCheck
VAR_INPUT
	Check : I_PreExecutionChecks;
END_VAR
VAR
	srcImageInfo : TcVnImageInfo;
	destImageInfo : TcVnImageInfo;
END_VAR
Check.IsTrue(ipSrcImage.IsValid, 'ipSrcImage must contain an image');

IF ipSrcImage.TryGetImageInfo(srcImageInfo) THEN
	Check.IsTrue((nSrcChannelIndex.Value <= srcImageInfo.stPixelFormat.nChannels), 'nSrcChannelIndex is greater than the available ipSrcImage channels');
END_IF

IF NOT ipDestImage.IsValid THEN
	RETURN;
END_IF

IF ipDestImage.TryGetImageInfo(destImageInfo) THEN
	Check.IsTrue((nDestChannelIndex.Value <= destImageInfo.stPixelFormat.nChannels), 'nDestChannelIndex is greater than the available ipDestImage channels');
END_IF

Check.IsTrue((srcImageInfo.nHeight = destImageInfo.nHeight), 'ipSrcImage must be the same height as ipDestImage');
Check.IsTrue((srcImageInfo.nWidth = destImageInfo.nWidth), 'ipSrcImage must be the same width as ipDestImage');
Check.IsTrue((srcImageInfo.stPixelFormat.nElementSize = destImageInfo.stPixelFormat.nElementSize), 'ipSrcImage  must have the same element size as ipDestImage');
END_METHOD

END_FUNCTION_BLOCK

// Nodes/Basic Image Ops/Node_F_VN_SetPixel
{attribute 'linkalways'} 
{attribute 'no_explicit_call' := 'This FB is a CLASS and must be accessed using methods or properties'}
{attribute 'enable_dynamic_creation'}
FUNCTION_BLOCK Node_F_VN_SetPixel EXTENDS VisionNode
VAR
    ipSrcImage : _ITcVnImage;
    aValue : _TcVnVector4_LREAL;
    nX : _UDINT(0);
    nY : _UDINT(0);
    hrPrev : _HRESULT(S_OK);
	hresult : _HRESULT(S_OK);
END_VAR

METHOD FB_init : BOOL
VAR_INPUT
	bInitRetains : BOOL; // if TRUE, the retain variables are initialized (warm start / cold start)
	bInCopyCode : BOOL;  // if TRUE, the instance afterwards gets moved into the copy code (online change)
END_VAR
AddInput('ipSrcImage', ipSrcImage);
AddInput('aValue', aValue);
AddParameter('nX', nX);
AddParameter('nY', nY);
AddInput('hrPrev', hrPrev);
AddOutput('hresult',hresult);
END_METHOD

METHOD PUBLIC  Clone : I_Node
VAR
	pNode : POINTER TO Node_F_VN_SetPixel;
END_VAR
pNode := __NEW(Node_F_VN_SetPixel);
Clone := pNode^;
END_METHOD

METHOD PROTECTED OnExecute
hresult.Value := F_VN_SetPixel(
    ipSrcImage := ipSrcImage.Value,
    aValue := aValue.Value,
    nX := nX.Value,
    nY := nY.Value,
	hrPrev:= hrPrev.Value);
END_METHOD

METHOD PUBLIC PreExecutionCheck
VAR_INPUT
	Check : I_PreExecutionChecks;
END_VAR
Check.IsTrue(ipSrcImage.IsValid, 'ipSrcImage must contain an image');
END_METHOD

END_FUNCTION_BLOCK

// Nodes/Basic Image Ops/Node_F_VN_SetPixels
{attribute 'linkalways'} 
{attribute 'no_explicit_call' := 'This FB is a CLASS and must be accessed using methods or properties'}
{attribute 'enable_dynamic_creation'}
FUNCTION_BLOCK Node_F_VN_SetPixels EXTENDS VisionNode
VAR
    ipDestImage : _ITcVnImage;
    aValue : _TcVnVector4_LREAL;
    hrPrev : _HRESULT(S_OK);
	hresult : _HRESULT(S_OK);
END_VAR

METHOD FB_init : BOOL
VAR_INPUT
	bInitRetains : BOOL; // if TRUE, the retain variables are initialized (warm start / cold start)
	bInCopyCode : BOOL;  // if TRUE, the instance afterwards gets moved into the copy code (online change)
END_VAR
AddInput('ipDestImage', ipDestImage);
AddInput('aValue', aValue);
AddInput('hrPrev', hrPrev);
AddOutput('ipDestImage', ipDestImage);
AddOutput('hresult',hresult);
END_METHOD

METHOD PUBLIC  Clone : I_Node
VAR
	pNode : POINTER TO Node_F_VN_SetPixels;
END_VAR
pNode := __NEW(Node_F_VN_SetPixels);
Clone := pNode^;
END_METHOD

METHOD PROTECTED OnExecute
hresult.Value := F_VN_SetPixels(
    ipDestImage := ipDestImage.Value,
    aValue := aValue.Value,
	hrPrev:= hrPrev.Value);
END_METHOD

METHOD PUBLIC PreExecutionCheck
VAR_INPUT
	Check : I_PreExecutionChecks;
END_VAR
Check.IsTrue(ipDestImage.IsValid, 'ipDestImage must contain an image');
END_METHOD

END_FUNCTION_BLOCK

// Nodes/Basic Image Ops/Node_F_VN_SetPixelsExp
{attribute 'linkalways'} 
{attribute 'no_explicit_call' := 'This FB is a CLASS and must be accessed using methods or properties'}
{attribute 'enable_dynamic_creation'}
FUNCTION_BLOCK Node_F_VN_SetPixelsExp EXTENDS VisionNode
VAR
    ipDestImage : _ITcVnImage;
    aValue : _TcVnVector4_LREAL;
    ipMask : _ITcVnImage;
    hrPrev : _HRESULT(S_OK);
	hresult : _HRESULT(S_OK);
END_VAR

METHOD FB_init : BOOL
VAR_INPUT
	bInitRetains : BOOL; // if TRUE, the retain variables are initialized (warm start / cold start)
	bInCopyCode : BOOL;  // if TRUE, the instance afterwards gets moved into the copy code (online change)
END_VAR
AddInput('ipDestImage', ipDestImage);
AddInput('aValue', aValue);
AddInput('ipMask', ipMask);
AddInput('hrPrev', hrPrev);
AddOutput('ipDestImage', ipDestImage);
AddOutput('hresult',hresult);
END_METHOD

METHOD PUBLIC  Clone : I_Node
VAR
	pNode : POINTER TO Node_F_VN_SetPixelsExp;
END_VAR
pNode := __NEW(Node_F_VN_SetPixelsExp);
Clone := pNode^;
END_METHOD

METHOD PROTECTED OnExecute
hresult.Value := F_VN_SetPixelsExp(
    ipDestImage := ipDestImage.Value,
    aValue := aValue.Value,
    ipMask := ipMask.Value,
	hrPrev:= hrPrev.Value);
END_METHOD

METHOD PUBLIC PreExecutionCheck
VAR_INPUT
	Check : I_PreExecutionChecks;
END_VAR
Check.IsTrue(ipDestImage.IsValid, 'ipDestImage must contain an image');
Check.IsTrue(ipMask.IsValid, 'ipMask must contain an image');
Check.IsTrue(ipMask.HasChannelCount(1), 'ipMask must have 1 channel');
Check.IsTrue(ipMask.IsPixelDepth(8), 'ipMask must have 8 bit pixel depth');
Check.IsTrue(IsImage1SizeEqualToImage2Size(ipMask.Value, ipDestImage.Value), 'ipMask must be the same size as ipDestImage');
END_METHOD

END_FUNCTION_BLOCK

// Nodes/Basic Image Ops/Node_F_VN_SetRoi
{attribute 'linkalways'} 
{attribute 'no_explicit_call' := 'This FB is a CLASS and must be accessed using methods or properties'}
{attribute 'enable_dynamic_creation'}
FUNCTION_BLOCK Node_F_VN_SetRoi EXTENDS VisionNode
VAR
    nX : _UDINT(0);
    nY : _UDINT(0);
    nWidth : _UDINT(0);
    nHeight : _UDINT(0);
    ipDestImage : _ITcVnImage;
    hrPrev : _HRESULT(S_OK);
	hresult : _HRESULT(S_OK);
END_VAR

METHOD FB_init : BOOL
VAR_INPUT
	bInitRetains : BOOL; // if TRUE, the retain variables are initialized (warm start / cold start)
	bInCopyCode : BOOL;  // if TRUE, the instance afterwards gets moved into the copy code (online change)
END_VAR
AddParameter('nX', nX);
AddParameter('nY', nY);
AddParameter('nWidth', nWidth);
AddParameter('nHeight', nHeight);
AddInput('ipDestImage', ipDestImage);
AddInput('hrPrev', hrPrev);
AddOutput('ipDestImage', ipDestImage);
AddOutput('hresult',hresult);
END_METHOD

METHOD PUBLIC  Clone : I_Node
VAR
	pNode : POINTER TO Node_F_VN_SetRoi;
END_VAR
pNode := __NEW(Node_F_VN_SetRoi);
Clone := pNode^;
END_METHOD

METHOD PROTECTED OnExecute
hresult.Value := F_VN_SetRoi(
    nX := nX.Value,
    nY := nY.Value,
    nWidth := nWidth.Value,
	nHeight := nHeight.Value,
	ipDestImage := ipDestImage.Value,
	hrPrev:= hrPrev.Value);
END_METHOD

METHOD PUBLIC PreExecutionCheck
VAR_INPUT
	Check : I_PreExecutionChecks;
END_VAR
VAR
    imgWidth : UDINT;
    imgHeight : UDINT;
    roiRectangle : TcVnRectangle_UDINT;
END_VAR
Check.IsTrue(ipDestImage.IsValid, 'ipDestImage must contain an image');

IF Check.Failed THEN
    RETURN;
END_IF

ipDestImage.Value.GetWidth(imgWidth);
ipDestImage.Value.GetHeight(imgHeight);
roiRectangle.nX := nX.Value;
roiRectangle.nY := nY.Value;
roiRectangle.nWidth := nWidth.Value;
roiRectangle.nHeight := nHeight.Value;

Check.IsTrue(IsRoiSizeOK_Udint(roiRectangle, imgWidth, imgHeight), 'ROI must fit within image');
END_METHOD

END_FUNCTION_BLOCK

// Nodes/Basic Image Ops/Node_F_VN_SetRoi_TcVnRectangle_DINT
{attribute 'linkalways'} 
{attribute 'no_explicit_call' := 'This FB is a CLASS and must be accessed using methods or properties'}
{attribute 'enable_dynamic_creation'}
FUNCTION_BLOCK Node_F_VN_SetRoi_TcVnRectangle_DINT EXTENDS VisionNode
VAR
    stRoi : _TcVnRectangle_DINT;
    ipDestImage : _ITcVnImage;
    hrPrev : _HRESULT(S_OK);
	hresult : _HRESULT(S_OK);
END_VAR

METHOD FB_init : BOOL
VAR_INPUT
	bInitRetains : BOOL; // if TRUE, the retain variables are initialized (warm start / cold start)
	bInCopyCode : BOOL;  // if TRUE, the instance afterwards gets moved into the copy code (online change)
END_VAR
AddInput('stRoi', stRoi);
AddInput('ipDestImage', ipDestImage);
AddInput('hrPrev', hrPrev);
AddOutput('ipDestImage', ipDestImage);
AddOutput('hresult',hresult);
END_METHOD

METHOD PUBLIC  Clone : I_Node
VAR
	pNode : POINTER TO Node_F_VN_SetRoi_TcVnRectangle_DINT;
END_VAR
pNode := __NEW(Node_F_VN_SetRoi_TcVnRectangle_DINT);
Clone := pNode^;
END_METHOD

METHOD PROTECTED OnExecute
hresult.Value := F_VN_SetRoi_TcVnRectangle_DINT(
    stRoi := stRoi.Value,
	ipDestImage := ipDestImage.Value,
	hrPrev:= hrPrev.Value);
END_METHOD

METHOD PUBLIC PreExecutionCheck
VAR_INPUT
	Check : I_PreExecutionChecks;
END_VAR
VAR
    imageWidth : UDINT;
    imageHeight : UDINT;
END_VAR
Check.IsTrue(ipDestImage.IsValid, 'ipDestImage must contain an image');

IF Check.Failed THEN
    RETURN;
END_IF

ipDestImage.Value.GetWidth(imageWidth);
ipDestImage.Value.GetHeight(imageHeight);

Check.IsTrue(IsRoiSizeOK_Dint(stRoi.Value, imageWidth, imageHeight), 'ROI must fit within image');
END_METHOD

END_FUNCTION_BLOCK

// Nodes/Basic Image Ops/Node_F_VN_SetRoi_TcVnRectangle_UDINT
{attribute 'linkalways'} 
{attribute 'no_explicit_call' := 'This FB is a CLASS and must be accessed using methods or properties'}
{attribute 'enable_dynamic_creation'}
FUNCTION_BLOCK Node_F_VN_SetRoi_TcVnRectangle_UDINT EXTENDS VisionNode
VAR
    stRoi : _TcVnRectangle_UDINT;
    ipDestImage : _ITcVnImage;
    hrPrev : _HRESULT(S_OK);
	hresult : _HRESULT(S_OK);
END_VAR

METHOD FB_init : BOOL
VAR_INPUT
	bInitRetains : BOOL; // if TRUE, the retain variables are initialized (warm start / cold start)
	bInCopyCode : BOOL;  // if TRUE, the instance afterwards gets moved into the copy code (online change)
END_VAR
AddInput('stRoi', stRoi);
AddInput('ipDestImage', ipDestImage);
AddInput('hrPrev', hrPrev);
AddOutput('ipDestImage', ipDestImage);
AddOutput('hresult',hresult);
END_METHOD

METHOD PUBLIC  Clone : I_Node
VAR
	pNode : POINTER TO Node_F_VN_SetRoi_TcVnRectangle_UDINT;
END_VAR
pNode := __NEW(Node_F_VN_SetRoi_TcVnRectangle_UDINT);
Clone := pNode^;
END_METHOD

METHOD PROTECTED OnExecute
hresult.Value := F_VN_SetRoi_TcVnRectangle_UDINT(
    stRoi := stRoi.Value,
	ipDestImage := ipDestImage.Value,
	hrPrev:= hrPrev.Value);
END_METHOD

METHOD PUBLIC PreExecutionCheck
VAR_INPUT
	Check : I_PreExecutionChecks;
END_VAR
VAR
    imageWidth : UDINT;
    imageHeight : UDINT;
END_VAR
Check.IsTrue(ipDestImage.IsValid, 'ipDestImage must contain an image');

IF Check.Failed THEN
    RETURN;
END_IF

ipDestImage.Value.GetWidth(imageWidth);
ipDestImage.Value.GetHeight(imageHeight);

Check.IsTrue(IsRoiSizeOK_Udint(stRoi.Value, imageWidth, imageHeight), 'ROI must fit within image');
END_METHOD

END_FUNCTION_BLOCK

// Nodes/Basic Image Ops/Node_F_VN_TransformIntoDisplayableImage
{attribute 'linkalways'} 
{attribute 'no_explicit_call' := 'This FB is a CLASS and must be accessed using methods or properties'}
{attribute 'enable_dynamic_creation'}
FUNCTION_BLOCK Node_F_VN_TransformIntoDisplayableImage EXTENDS VisionNode
VAR
    ipSrcImage : _ITcVnImage;
    ipDestImage : _ITcVnDisplayableImage;
    hrPrev : _HRESULT(S_OK);
	hresult : _HRESULT(S_OK);
END_VAR

METHOD FB_init : BOOL
VAR_INPUT
	bInitRetains : BOOL; // if TRUE, the retain variables are initialized (warm start / cold start)
	bInCopyCode : BOOL;  // if TRUE, the instance afterwards gets moved into the copy code (online change)
END_VAR
AddInput('ipSrcImage', ipSrcImage);
AddInput('hrPrev', hrPrev);
AddOutput('ipDestImage', ipDestImage);
AddOutput('hresult',hresult);
END_METHOD

METHOD PUBLIC  Clone : I_Node
VAR
	pNode : POINTER TO Node_F_VN_TransformIntoDisplayableImage;
END_VAR
pNode := __NEW(Node_F_VN_TransformIntoDisplayableImage);
Clone := pNode^;
END_METHOD

METHOD PROTECTED OnExecute
hresult.Value := F_VN_TransformIntoDisplayableImage(
    ipSrcImage := ipSrcImage.Value,
	ipDestImage := ipDestImage.Value,
	hrPrev:= hrPrev.Value);
END_METHOD

METHOD PUBLIC PreExecutionCheck
VAR_INPUT
	Check : I_PreExecutionChecks;
END_VAR
Check.IsTrue(ipSrcImage.IsValid, 'ipSrcImage must contain an image');
END_METHOD

END_FUNCTION_BLOCK

// Nodes/Basic Image Ops/Node_F_VN_TransformIntoDisplayableImageExp
{attribute 'linkalways'} 
{attribute 'no_explicit_call' := 'This FB is a CLASS and must be accessed using methods or properties'}
{attribute 'enable_dynamic_creation'}
FUNCTION_BLOCK Node_F_VN_TransformIntoDisplayableImageExp EXTENDS VisionNode
VAR
    ipSrcImage : _ITcVnImage;
    ipDestImage : _ITcVnDisplayableImage;
    bAllowDeepCopy : _BOOL(FALSE);
    hrPrev : _HRESULT(S_OK);
	hresult : _HRESULT(S_OK);
END_VAR

METHOD FB_init : BOOL
VAR_INPUT
	bInitRetains : BOOL; // if TRUE, the retain variables are initialized (warm start / cold start)
	bInCopyCode : BOOL;  // if TRUE, the instance afterwards gets moved into the copy code (online change)
END_VAR
AddInput('ipSrcImage', ipSrcImage);
AddParameter('bAllowDeepCopy', bAllowDeepCopy);
AddInput('hrPrev', hrPrev);
AddOutput('ipDestImage', ipDestImage);
AddOutput('hresult',hresult);
END_METHOD

METHOD PUBLIC  Clone : I_Node
VAR
	pNode : POINTER TO Node_F_VN_TransformIntoDisplayableImageExp;
END_VAR
pNode := __NEW(Node_F_VN_TransformIntoDisplayableImageExp);
Clone := pNode^;
END_METHOD

METHOD PROTECTED OnExecute
hresult.Value := F_VN_TransformIntoDisplayableImageExp(
    ipSrcImage := ipSrcImage.Value,
    bAllowDeepCopy := bAllowDeepCopy.Value,
	ipDestImage := ipDestImage.Value,
	hrPrev:= hrPrev.Value);
END_METHOD

METHOD PUBLIC PreExecutionCheck
VAR_INPUT
	Check : I_PreExecutionChecks;
END_VAR
Check.IsTrue(ipSrcImage.IsValid, 'ipSrcImage must contain an image');
END_METHOD

END_FUNCTION_BLOCK

// Nodes/Code Quality/Node_F_VN_GradeBarcode
{attribute 'linkalways'} 
{attribute 'no_explicit_call' := 'This FB is a CLASS and must be accessed using methods or properties'}
{attribute 'enable_dynamic_creation'}
FUNCTION_BLOCK Node_F_VN_GradeBarcode EXTENDS VisionNode
VAR
    ipSrcImage : _ITcVnImage;
    ipDecodedData : _ITcVnContainer;
    stCodeGrades : 	_TcVnCodeGrades1D;
    eBarcodeType : _ETcVnBarcodeType(ETcVnBarcodeType.TCVN_BT_ANY);
    fAngleDeg : _REAL(0.0);
    hrPrev : _HRESULT(S_OK);
	hresult : _HRESULT(S_OK);
END_VAR

METHOD FB_init : BOOL
VAR_INPUT
	bInitRetains : BOOL; // if TRUE, the retain variables are initialized (warm start / cold start)
	bInCopyCode : BOOL;  // if TRUE, the instance afterwards gets moved into the copy code (online change)
END_VAR
AddInput('ipSrcImage', ipSrcImage);
AddParameter('eBarcodeType', eBarcodeType);
AddInput('hrPrev', hrPrev);
AddOutput('ipDecodedData', ipDecodedData);
AddOutput('stCodeGrades', stCodeGrades);
AddOutput('fAngleDeg', fAngleDeg);
AddOutput('hresult', hresult);
END_METHOD

METHOD PUBLIC  Clone : I_Node
VAR
	pNode : POINTER TO Node_F_VN_GradeBarcode;
END_VAR
pNode := __NEW(Node_F_VN_GradeBarcode);
Clone := pNode^;
END_METHOD

METHOD PROTECTED OnExecute
VAR
    angle : REAL;
END_VAR
hresult.Value := F_VN_GradeBarcode(
	ipSrcImage := ipSrcImage.Value,
    ipDecodedData := ipDecodedData.Value,
    stCodeGrades := stCodeGrades.Value,
    eBarcodeType := eBarcodeType.Value,
	hrPrev:= hrPrev.Value,
    fAngleDeg => angle);

fAngleDeg.Value := angle;
END_METHOD

METHOD PUBLIC PreExecutionCheck
VAR_INPUT
	Check : I_PreExecutionChecks;
END_VAR
VAR
    barcodeTypeIsValid : BOOL;
END_VAR
Check.IsTrue(ipSrcImage.IsValid, 'ipSrcImage must contain an image');
Check.IsTrue(ipSrcImage.HasChannelCount(1), 'ipSrcImage must have 1 channel');
Check.IsTrue(ipSrcImage.IsPixelDepth(8), 'ipSrcImage must have 8 bit pixel depth');

CASE eBarcodeType.Value OF
    ETcVnBarcodeType.TCVN_BT_CODE39,
    ETcVnBarcodeType.TCVN_BT_CODE128,
    ETcVnBarcodeType.TCVN_BT_EAN8,
    ETcVnBarcodeType.TCVN_BT_EAN13,
    ETcVnBarcodeType.TCVN_BT_ITF,
    ETcVnBarcodeType.TCVN_BT_UPCA,
    ETcVnBarcodeType.TCVN_BT_UPCE :
        barcodeTypeIsValid := TRUE;
END_CASE

Check.IsTrue(barcodeTypeIsValid, 'eBarcodeType must have supported type');
END_METHOD

END_FUNCTION_BLOCK

// Nodes/Code Quality/Node_F_VN_GradeBarcodeExp
{attribute 'linkalways'} 
{attribute 'no_explicit_call' := 'This FB is a CLASS and must be accessed using methods or properties'}
{attribute 'enable_dynamic_creation'}
FUNCTION_BLOCK Node_F_VN_GradeBarcodeExp EXTENDS VisionNode
VAR
    ipSrcImage : _ITcVnImage;
    ipDecodedData : _ITcVnContainer;
    stCodeGrades : 	_TcVnCodeGrades1D;
    eBarcodeType : _ETcVnBarcodeType(ETcVnBarcodeType.TCVN_BT_ANY);
    eSearchDirection : _ETcVnBarcodeSearchDirection(ETcVnBarcodeSearchDirection.TCVN_BSD_ANY);
    ipResultVisualization : _ITcVnImage;
    ipScanLineInfo : _ITcVnContainer;
    ipContour : _ITcVnContainer;
    fAngleDeg : _REAL(0.0);
    hrPrev : _HRESULT(S_OK);
	hresult : _HRESULT(S_OK);
END_VAR

METHOD FB_init : BOOL
VAR_INPUT
	bInitRetains : BOOL; // if TRUE, the retain variables are initialized (warm start / cold start)
	bInCopyCode : BOOL;  // if TRUE, the instance afterwards gets moved into the copy code (online change)
END_VAR
AddInput('ipSrcImage', ipSrcImage);
AddParameter('eBarcodeType', eBarcodeType);
AddParameter('eSearchDirection', eSearchDirection);
AddInput('hrPrev', hrPrev);
AddOutput('ipDecodedData', ipDecodedData);
AddOutput('stCodeGrades', stCodeGrades);
AddOutput('ipResultVisualization', ipResultVisualization);
AddOutput('ipScanLineInfo', ipScanLineInfo);
AddOutput('ipContour', ipContour);
AddOutput('fAngleDeg', fAngleDeg);
AddOutput('hresult', hresult);
END_METHOD

METHOD PUBLIC  Clone : I_Node
VAR
	pNode : POINTER TO Node_F_VN_GradeBarcodeExp;
END_VAR
pNode := __NEW(Node_F_VN_GradeBarcodeExp);
Clone := pNode^;
END_METHOD

METHOD PROTECTED OnExecute
VAR
    angle : REAL;
END_VAR
hresult.Value := F_VN_GradeBarcodeExp(
	ipSrcImage := ipSrcImage.Value,
    ipDecodedData := ipDecodedData.Value,
    stCodeGrades := stCodeGrades.Value,
    eBarcodeType := eBarcodeType.Value,
    eSearchDirection := eSearchDirection.Value,
    ipResultVisualization := ipResultVisualization.Value,
    ipScanLineInfo := ipScanLineInfo.Value,
    ipContour := ipContour.Value,
	hrPrev:= hrPrev.Value,
    fAngleDeg => angle);

fAngleDeg.Value := angle;
END_METHOD

METHOD PUBLIC PreExecutionCheck
VAR_INPUT
	Check : I_PreExecutionChecks;
END_VAR
VAR
    barcodeTypeIsValid : BOOL;
END_VAR
Check.IsTrue(ipSrcImage.IsValid, 'ipSrcImage must contain an image');
Check.IsTrue(ipSrcImage.HasChannelCount(1), 'ipSrcImage must have 1 channel');
Check.IsTrue(ipSrcImage.IsPixelDepth(8), 'ipSrcImage must have 8 bit pixel depth');

CASE eBarcodeType.Value OF
    ETcVnBarcodeType.TCVN_BT_CODE39,
    ETcVnBarcodeType.TCVN_BT_CODE128,
    ETcVnBarcodeType.TCVN_BT_EAN8,
    ETcVnBarcodeType.TCVN_BT_EAN13,
    ETcVnBarcodeType.TCVN_BT_ITF,
    ETcVnBarcodeType.TCVN_BT_UPCA,
    ETcVnBarcodeType.TCVN_BT_UPCE :
        barcodeTypeIsValid := TRUE;
END_CASE

Check.IsTrue(barcodeTypeIsValid, 'eBarcodeType must have supported type');
END_METHOD

END_FUNCTION_BLOCK

// Nodes/Code Quality/Node_F_VN_GradeDataMatrixCode
{attribute 'linkalways'} 
{attribute 'no_explicit_call' := 'This FB is a CLASS and must be accessed using methods or properties'}
{attribute 'enable_dynamic_creation'}
FUNCTION_BLOCK Node_F_VN_GradeDataMatrixCode EXTENDS VisionNode
VAR
    ipSrcImage : _ITcVnImage;
    ipDecodedData : _ITcVnContainer;
    stCodeGrades : 	_TcVnCodeGradesDM;
    fModuleWidth : _REAL(4.0);
    fAngleDeg : _REAL(0.0);
    hrPrev : _HRESULT(S_OK);
	hresult : _HRESULT(S_OK);
END_VAR

METHOD FB_init : BOOL
VAR_INPUT
	bInitRetains : BOOL; // if TRUE, the retain variables are initialized (warm start / cold start)
	bInCopyCode : BOOL;  // if TRUE, the instance afterwards gets moved into the copy code (online change)
END_VAR
AddInput('ipSrcImage', ipSrcImage);
AddParameter('fModuleWidth', fModuleWidth);
AddInput('hrPrev', hrPrev);
AddOutput('ipDecodedData', ipDecodedData);
AddOutput('stCodeGrades', stCodeGrades);
AddOutput('fAngleDeg', fAngleDeg);
AddOutput('hresult', hresult);
END_METHOD

METHOD PUBLIC  Clone : I_Node
VAR
	pNode : POINTER TO Node_F_VN_GradeDataMatrixCode;
END_VAR
pNode := __NEW(Node_F_VN_GradeDataMatrixCode);
Clone := pNode^;
END_METHOD

METHOD PROTECTED OnExecute
VAR
    angle : REAL;
END_VAR
hresult.Value := F_VN_GradeDataMatrixCode(
	ipSrcImage := ipSrcImage.Value,
    ipDecodedData := ipDecodedData.Value,
    stCodeGrades := stCodeGrades.Value,
    fModuleWidth := fModuleWidth.Value,
	hrPrev:= hrPrev.Value,
    fAngleDeg => angle);

fAngleDeg.Value := angle;
END_METHOD

METHOD PUBLIC PreExecutionCheck
VAR_INPUT
	Check : I_PreExecutionChecks;
END_VAR
Check.IsTrue(ipSrcImage.IsValid, 'ipSrcImage must contain an image');
Check.IsTrue(ipSrcImage.HasChannelCount(1), 'ipSrcImage must have 1 channel');
Check.IsTrue(ipSrcImage.IsPixelDepth(8), 'ipSrcImage must have 8 bit pixel depth');
Check.IsTrue(fModuleWidth.Value >= 3, 'fModuleWidth must be greater than or equal to 3');
END_METHOD

END_FUNCTION_BLOCK

// Nodes/Code Quality/Node_F_VN_GradeDataMatrixCodeExp
{attribute 'linkalways'} 
{attribute 'no_explicit_call' := 'This FB is a CLASS and must be accessed using methods or properties'}
{attribute 'enable_dynamic_creation'}
FUNCTION_BLOCK Node_F_VN_GradeDataMatrixCodeExp EXTENDS VisionNode
VAR
    ipSrcImage : _ITcVnImage;
    ipDecodedData : _ITcVnContainer;
    stCodeGrades : 	_TcVnCodeGradesDM;
    fModuleWidth : _REAL(4.0);
    ipResultVisualization : _ITcVnImage;
    ipMarginGrades : _ITcVnContainer;
    ipContour : _ITcVnContainer;
    fAngleDeg : _REAL(0.0);
    hrPrev : _HRESULT(S_OK);
	hresult : _HRESULT(S_OK);
END_VAR

METHOD FB_init : BOOL
VAR_INPUT
	bInitRetains : BOOL; // if TRUE, the retain variables are initialized (warm start / cold start)
	bInCopyCode : BOOL;  // if TRUE, the instance afterwards gets moved into the copy code (online change)
END_VAR
AddInput('ipSrcImage', ipSrcImage);
AddParameter('fModuleWidth', fModuleWidth);
AddInput('hrPrev', hrPrev);
AddOutput('ipDecodedData', ipDecodedData);
AddOutput('stCodeGrades', stCodeGrades);
AddOutput('ipResultVisualization', ipResultVisualization);
AddOutput('ipMarginGrades', ipMarginGrades);
AddOutput('ipContour', ipContour);
AddOutput('fAngleDeg', fAngleDeg);
AddOutput('hresult', hresult);
END_METHOD

METHOD PUBLIC  Clone : I_Node
VAR
	pNode : POINTER TO Node_F_VN_GradeDataMatrixCodeExp;
END_VAR
pNode := __NEW(Node_F_VN_GradeDataMatrixCodeExp);
Clone := pNode^;
END_METHOD

METHOD PROTECTED OnExecute
VAR
    angle : REAL;
END_VAR
hresult.Value := F_VN_GradeDataMatrixCodeExp(
	ipSrcImage := ipSrcImage.Value,
    ipDecodedData := ipDecodedData.Value,
    stCodeGrades := stCodeGrades.Value,
    fModuleWidth := fModuleWidth.Value,
    ipResultVisualization := ipResultVisualization.Value,
    ipMarginGrades := ipMarginGrades.Value,
    ipContour := ipContour.Value,
	hrPrev:= hrPrev.Value,
    fAngleDeg => angle);

fAngleDeg.Value := angle;
END_METHOD

METHOD PUBLIC PreExecutionCheck
VAR_INPUT
	Check : I_PreExecutionChecks;
END_VAR
Check.IsTrue(ipSrcImage.IsValid, 'ipSrcImage must contain an image');
Check.IsTrue(ipSrcImage.HasChannelCount(1), 'ipSrcImage must have 1 channel');
Check.IsTrue(ipSrcImage.IsPixelDepth(8), 'ipSrcImage must have 8 bit pixel depth');
Check.IsTrue(fModuleWidth.Value >= 3, 'fModuleWidth must be greater than or equal to 3');
END_METHOD

END_FUNCTION_BLOCK

// Nodes/Code Quality/Node_F_VN_GradeQRCode
{attribute 'linkalways'} 
{attribute 'no_explicit_call' := 'This FB is a CLASS and must be accessed using methods or properties'}
{attribute 'enable_dynamic_creation'}
FUNCTION_BLOCK Node_F_VN_GradeQRCode EXTENDS VisionNode
VAR
    ipSrcImage : _ITcVnImage;
    ipDecodedData : _ITcVnContainer;
    stCodeGrades : 	_TcVnCodeGradesQR;
    fModuleWidth : _REAL(4.0);
    fAngleDeg : _REAL(0.0);
    hrPrev : _HRESULT(S_OK);
	hresult : _HRESULT(S_OK);
END_VAR

METHOD FB_init : BOOL
VAR_INPUT
	bInitRetains : BOOL; // if TRUE, the retain variables are initialized (warm start / cold start)
	bInCopyCode : BOOL;  // if TRUE, the instance afterwards gets moved into the copy code (online change)
END_VAR
AddInput('ipSrcImage', ipSrcImage);
AddParameter('fModuleWidth', fModuleWidth);
AddInput('hrPrev', hrPrev);
AddOutput('ipDecodedData', ipDecodedData);
AddOutput('stCodeGrades', stCodeGrades);
AddOutput('fAngleDeg', fAngleDeg);
AddOutput('hresult', hresult);
END_METHOD

METHOD PUBLIC  Clone : I_Node
VAR
	pNode : POINTER TO Node_F_VN_GradeQRCode;
END_VAR
pNode := __NEW(Node_F_VN_GradeQRCode);
Clone := pNode^;
END_METHOD

METHOD PROTECTED OnExecute
VAR
    angle : REAL;
END_VAR
hresult.Value := F_VN_GradeQRCode(
	ipSrcImage := ipSrcImage.Value,
    ipDecodedData := ipDecodedData.Value,
    stCodeGrades := stCodeGrades.Value,
    fModuleWidth := fModuleWidth.Value,
	hrPrev:= hrPrev.Value,
    fAngleDeg => angle);
    
fAngleDeg.Value := angle;
END_METHOD

METHOD PUBLIC PreExecutionCheck
VAR_INPUT
	Check : I_PreExecutionChecks;
END_VAR
Check.IsTrue(ipSrcImage.IsValid, 'ipSrcImage must contain an image');
Check.IsTrue(ipSrcImage.HasChannelCount(1), 'ipSrcImage must have 1 channel');
Check.IsTrue(ipSrcImage.IsPixelDepth(8), 'ipSrcImage must have 8 bit pixel depth');
Check.IsTrue(fModuleWidth.Value >= 3, 'fModuleWidth must be greater than or equal to 3');
END_METHOD

END_FUNCTION_BLOCK

// Nodes/Code Quality/Node_F_VN_GradeQRCodeExp
{attribute 'linkalways'} 
{attribute 'no_explicit_call' := 'This FB is a CLASS and must be accessed using methods or properties'}
{attribute 'enable_dynamic_creation'}
FUNCTION_BLOCK Node_F_VN_GradeQRCodeExp EXTENDS VisionNode
VAR
    ipSrcImage : _ITcVnImage;
    ipDecodedData : _ITcVnContainer;
    stCodeGrades : 	_TcVnCodeGradesQR;
    fModuleWidth : _REAL(4.0);
    ipResultVisualization : _ITcVnImage;
    ipMarginGrades : _ITcVnContainer;
    ipContour : _ITcVnContainer;
    fAngleDeg : _REAL(0.0);
    hrPrev : _HRESULT(S_OK);
	hresult : _HRESULT(S_OK);
END_VAR

METHOD FB_init : BOOL
VAR_INPUT
	bInitRetains : BOOL; // if TRUE, the retain variables are initialized (warm start / cold start)
	bInCopyCode : BOOL;  // if TRUE, the instance afterwards gets moved into the copy code (online change)
END_VAR
AddInput('ipSrcImage', ipSrcImage);
AddParameter('fModuleWidth', fModuleWidth);
AddInput('hrPrev', hrPrev);
AddOutput('ipDecodedData', ipDecodedData);
AddOutput('stCodeGrades', stCodeGrades);
AddOutput('ipResultVisualization', ipResultVisualization);
AddOutput('ipMarginGrades', ipMarginGrades);
AddOutput('ipContour', ipContour);
AddOutput('fAngleDeg', fAngleDeg);
AddOutput('hresult', hresult);
END_METHOD

METHOD PUBLIC  Clone : I_Node
VAR
	pNode : POINTER TO Node_F_VN_GradeQRCodeExp;
END_VAR
pNode := __NEW(Node_F_VN_GradeQRCodeExp);
Clone := pNode^;
END_METHOD

METHOD PROTECTED OnExecute
VAR
    angle : REAL;
END_VAR
hresult.Value := F_VN_GradeQRCodeExp(
	ipSrcImage := ipSrcImage.Value,
    ipDecodedData := ipDecodedData.Value,
    stCodeGrades := stCodeGrades.Value,
    fModuleWidth := fModuleWidth.Value,
    ipResultVisualization := ipResultVisualization.Value,
    ipMarginGrades := ipMarginGrades.Value,
    ipContour := ipContour.Value,
	hrPrev:= hrPrev.Value,
    fAngleDeg => angle);
    
fAngleDeg.Value := angle;
END_METHOD

METHOD PUBLIC PreExecutionCheck
VAR_INPUT
	Check : I_PreExecutionChecks;
END_VAR
Check.IsTrue(ipSrcImage.IsValid, 'ipSrcImage must contain an image');
Check.IsTrue(ipSrcImage.HasChannelCount(1), 'ipSrcImage must have 1 channel');
Check.IsTrue(ipSrcImage.IsPixelDepth(8), 'ipSrcImage must have 8 bit pixel depth');
Check.IsTrue(fModuleWidth.Value >= 3, 'fModuleWidth must be greater than or equal to 3');
END_METHOD

END_FUNCTION_BLOCK

// Nodes/Code Reading/Node_F_VN_AnalyzeBarcodeWalsh
{attribute 'linkalways'}
{attribute 'no_explicit_call' := 'This FB is a CLASS and must be accessed using methods or properties'}
{attribute 'enable_dynamic_creation'}
FUNCTION_BLOCK Node_F_VN_AnalyzeBarcodeWalsh EXTENDS VisionNode
VAR
    ipBarcodeImage : _ITcVnImage;
    stParams : _TcVnParamsWalshBarcodeDetection;
    hrPrev : _HRESULT(S_OK);
    hresult : _HRESULT(S_OK);
END_VAR

METHOD FB_init : BOOL
VAR_INPUT
    bInitRetains : BOOL;
    bInCopyCode : BOOL;
END_VAR
AddInput('ipBarcodeImage', ipBarcodeImage);
AddInput('stParams', stParams);
AddInput('hrPrev', hrPrev);
AddOutput('stParams', stParams);
AddOutput('hresult', hresult);
END_METHOD

METHOD PUBLIC Clone : I_Node
VAR
    pNode : POINTER TO Node_F_VN_AnalyzeBarcodeWalsh;
END_VAR
pNode := __NEW(Node_F_VN_AnalyzeBarcodeWalsh);
Clone := pNode^;
END_METHOD

METHOD PROTECTED OnExecute
hresult.Value := F_VN_AnalyzeBarcodeWalsh(
    ipBarcodeImage := ipBarcodeImage.Value,
    stParams := stParams.Value,
    hrPrev := hrPrev.Value);
END_METHOD

METHOD PUBLIC PreExecutionCheck
VAR_INPUT
    Check : I_PreExecutionChecks;
END_VAR
Check.IsTrue(ipBarcodeImage.IsValid, 'ipBarcodeImage must contain an image');
END_METHOD

END_FUNCTION_BLOCK

// Nodes/Code Reading/Node_F_VN_DetectBarcodesWalsh
{attribute 'linkalways'}
{attribute 'no_explicit_call' := 'This FB is a CLASS and must be accessed using methods or properties'}
{attribute 'enable_dynamic_creation'}
FUNCTION_BLOCK Node_F_VN_DetectBarcodesWalsh EXTENDS VisionNode
VAR
    ipSrcImage : _ITcVnImage;
    ipBarcodes : _ITcVnContainer;
    eOptions : _UDINT(ETcVnDetectBarcodesWalshOptions.TCVN_DBWO_HORIZONTAL);
    stParams : _TcVnParamsWalshBarcodeDetection;
    hrPrev : _HRESULT(S_OK);
    hresult : _HRESULT(S_OK);
END_VAR

METHOD FB_init : BOOL
VAR_INPUT
    bInitRetains : BOOL;
    bInCopyCode : BOOL;
END_VAR
AddInput('ipSrcImage', ipSrcImage);
AddOutput('ipBarcodes', ipBarcodes);
AddParameter('eOptions', eOptions);
AddInput('stParams', stParams);
AddInput('hrPrev', hrPrev);
AddOutput('hresult', hresult);
END_METHOD

METHOD PUBLIC Clone : I_Node
VAR
    pNode : POINTER TO Node_F_VN_DetectBarcodesWalsh;
END_VAR
pNode := __NEW(Node_F_VN_DetectBarcodesWalsh);
Clone := pNode^;
END_METHOD

METHOD PROTECTED OnExecute
hresult.Value := F_VN_DetectBarcodesWalsh(
    ipSrcImage := ipSrcImage.Value,
    ipBarcodes := ipBarcodes.Value,
    eOptions := eOptions.Value,
    stParams := stParams.Value,
    hrPrev := hrPrev.Value);
END_METHOD

METHOD PUBLIC PreExecutionCheck
VAR_INPUT
    Check : I_PreExecutionChecks;
END_VAR
Check.IsTrue(ipSrcImage.IsValid, 'ipSrcImage must contain an image');
Check.IsTrue(stParams.Value.nMaxBarDistance > 0, 'nMaxBarDistance must be greater than 0');
Check.IsTrue(stParams.Value.fMinAspectRatio > 0.0, 'fMinAspectRatio must be greater than 0');
Check.IsTrue(stParams.Value.fMaxAspectRatio >= stParams.Value.fMinAspectRatio, 'fMaxAspectRatio must be at least fMinAspectRatio');
// -1 selects the automatic guess derived from nMaxBarDistance.
Check.IsTrue((stParams.Value.nMinArea = -1) OR (stParams.Value.nMinArea > 0), 'nMinArea must be -1 for the automatic guess, or greater than 0');
// -1 selects automatic graylevel conversion.
Check.IsTrue(stParams.Value.nChannelIndex >= -1, 'nChannelIndex must be -1 for automatic graylevel conversion, or a channel index');
Check.IsTrue(stParams.Value.nWalshFilterNum > 0, 'nWalshFilterNum must be greater than 0');
Check.IsTrue(stParams.Value.fPostProcessingResizeFactor > 0.0, 'fPostProcessingResizeFactor must be greater than 0');
END_METHOD

END_FUNCTION_BLOCK

// Nodes/Code Reading/Node_F_VN_DetectCodesNeuralNetwork
{attribute 'linkalways'} 
{attribute 'no_explicit_call' := 'This FB is a CLASS and must be accessed using methods or properties'}
{attribute 'enable_dynamic_creation'}
FUNCTION_BLOCK Node_F_VN_DetectCodesNeuralNetwork EXTENDS VisionNode
VAR
    ipSrcImage : _ITcVnImage;
    ipCodeRegions : _ITcVnContainer;
    ipCodeTypes : _ITcVnContainer;
	eModelType : _ETcVnCodeDetectionModel(ETcVnCodeDetectionModel.TCVN_CDM_DETECT_1_1);
	nCodeType : _ULINT(0);
    hrPrev : _HRESULT(S_OK);
	hresult : _HRESULT(S_OK);
END_VAR

METHOD FB_init : BOOL
VAR_INPUT
	bInitRetains : BOOL; // if TRUE, the retain variables are initialized (warm start / cold start)
	bInCopyCode : BOOL;  // if TRUE, the instance afterwards gets moved into the copy code (online change)
END_VAR
AddInput('ipSrcImage', ipSrcImage);
AddInput('eModelType', eModelType);
AddInput('nCodeType', nCodeType);
AddInput('hrPrev', hrPrev);
AddOutput('ipCodeRegions', ipCodeRegions);
AddOutput('ipCodeTypes', ipCodeTypes);
AddOutput('hresult', hresult);
END_METHOD

METHOD PUBLIC  Clone : I_Node
VAR
	pNode : POINTER TO Node_F_VN_DetectCodesNeuralNetwork;
END_VAR
pNode := __NEW(Node_F_VN_DetectCodesNeuralNetwork);
Clone := pNode^;
END_METHOD

METHOD PROTECTED OnExecute
hresult.Value := F_VN_DetectCodesNeuralNetwork(
	ipSrcImage := ipSrcImage.Value,
	ipCodeRegions := ipCodeRegions.Value,
	ipCodeTypes := ipCodeTypes.Value,
    eModelType := eModelType.Value,
    nCodeType := nCodeType.Value,
	hrPrev:= hrPrev.Value
);
END_METHOD

METHOD PUBLIC PreExecutionCheck
VAR_INPUT
	Check : I_PreExecutionChecks;
END_VAR
Check.IsTrue(ipSrcImage.IsValid, 'ipSrcImage must contain an image');
Check.IsTrue((ipSrcImage.HasChannelCount(1) OR ipSrcImage.HasChannelCount(3)), 'ipSrcImage must contain 1 or 3 channels');
END_METHOD

END_FUNCTION_BLOCK

// Nodes/Code Reading/Node_F_VN_ReadBarcode
{attribute 'linkalways'} 
{attribute 'no_explicit_call' := 'This FB is a CLASS and must be accessed using methods or properties'}
{attribute 'enable_dynamic_creation'}
FUNCTION_BLOCK Node_F_VN_ReadBarcode EXTENDS VisionNode
VAR
    ipSrcImage : _ITcVnImage;
    ipDecodedData : _ITcVnContainer;
    eBarcodeType : _ETcVnBarcodeType(ETcVnBarcodeType.TCVN_BT_ANY);
    hrPrev : _HRESULT(S_OK);
	hresult : _HRESULT(S_OK);
END_VAR

METHOD FB_init : BOOL
VAR_INPUT
	bInitRetains : BOOL; // if TRUE, the retain variables are initialized (warm start / cold start)
	bInCopyCode : BOOL;  // if TRUE, the instance afterwards gets moved into the copy code (online change)
END_VAR
AddInput('ipSrcImage', ipSrcImage);
AddParameter('eBarcodeType', eBarcodeType);
AddInput('hrPrev', hrPrev);
AddOutput('ipDecodedData', ipDecodedData);
AddOutput('hresult',hresult);
END_METHOD

METHOD PUBLIC  Clone : I_Node
VAR
	pNode : POINTER TO Node_F_VN_ReadBarcode;
END_VAR
pNode := __NEW(Node_F_VN_ReadBarcode);
Clone := pNode^;
END_METHOD

METHOD PROTECTED OnExecute
hresult.Value := F_VN_ReadBarcode(
	ipSrcImage := ipSrcImage.Value,
    ipDecodedData := ipDecodedData.Value,
    eBarcodeType := eBarcodeType.Value,
	hrPrev:= hrPrev.Value);
END_METHOD

METHOD PUBLIC PreExecutionCheck
VAR_INPUT
	Check : I_PreExecutionChecks;
END_VAR
Check.IsTrue(ipSrcImage.IsValid, 'ipSrcImage must contain an image');
Check.IsTrue((ipSrcImage.HasChannelCount(1) OR ipSrcImage.HasChannelCount(3)), 'ipSrcImage must have 1 or 3 channels');
Check.IsTrue(ipSrcImage.IsPixelDepth(8), 'ipSrcImage must have 8 bit pixel depth');
END_METHOD

END_FUNCTION_BLOCK

// Nodes/Code Reading/Node_F_VN_ReadBarcodeExp
{attribute 'linkalways'} 
{attribute 'no_explicit_call' := 'This FB is a CLASS and must be accessed using methods or properties'}
{attribute 'enable_dynamic_creation'}
FUNCTION_BLOCK Node_F_VN_ReadBarcodeExp EXTENDS VisionNode
VAR
    ipSrcImage : _ITcVnImage;
    ipDecodedData : _ITcVnContainer;
	ipContours : _ITcVnContainer;
    eBarcodeType : _ETcVnBarcodeType(ETcVnBarcodeType.TCVN_BT_ANY);
	nCodeNumber : _DINT(1);
	eSearchDirection : _ETcVnBarcodeSearchDirection(ETcVnBarcodeSearchDirection.TCVN_BSD_ANY);
    hrPrev : _HRESULT(S_OK);
	hresult : _HRESULT(S_OK);
END_VAR

METHOD FB_init : BOOL
VAR_INPUT
	bInitRetains : BOOL; // if TRUE, the retain variables are initialized (warm start / cold start)
	bInCopyCode : BOOL;  // if TRUE, the instance afterwards gets moved into the copy code (online change)
END_VAR
AddInput('ipSrcImage', ipSrcImage);
AddParameter('eBarcodeType', eBarcodeType);
AddParameter('nCodeNumber', nCodeNumber);
AddParameter('eSearchDirection', eSearchDirection);
AddInput('hrPrev', hrPrev);
AddOutput('ipDecodedData', ipDecodedData);
AddOutput('ipContours', ipContours);
AddOutput('hresult',hresult);
END_METHOD

METHOD PUBLIC  Clone : I_Node
VAR
	pNode : POINTER TO Node_F_VN_ReadBarcodeExp;
END_VAR
pNode := __NEW(Node_F_VN_ReadBarcodeExp);
Clone := pNode^;
END_METHOD

METHOD PROTECTED OnExecute
hresult.Value := F_VN_ReadBarcodeExp(
	ipSrcImage := ipSrcImage.Value,
    ipDecodedData := ipDecodedData.Value,
	ipContours := ipContours.Value,
    eBarcodeType := eBarcodeType.Value,
	nCodeNumber := nCodeNumber.Value,
	eSearchDirection := eSearchDirection.Value,
	hrPrev:= hrPrev.Value);
END_METHOD

METHOD PUBLIC PreExecutionCheck
VAR_INPUT
	Check : I_PreExecutionChecks;
END_VAR
Check.IsTrue(ipSrcImage.IsValid, 'ipSrcImage must contain an image');
Check.IsTrue((ipSrcImage.HasChannelCount(1) OR ipSrcImage.HasChannelCount(3)), 'ipSrcImage must have 1 or 3 channels');
Check.IsTrue(ipSrcImage.IsPixelDepth(8), 'ipSrcImage must have 8 bit pixel depth');
Check.IsTrue((nCodeNumber.Value = 1), 'nCodeNumber, currently only 1 supported');
END_METHOD

END_FUNCTION_BLOCK

// Nodes/Code Reading/Node_F_VN_ReadBarcodeExp2
{attribute 'linkalways'} 
{attribute 'no_explicit_call' := 'This FB is a CLASS and must be accessed using methods or properties'}
{attribute 'enable_dynamic_creation'}
FUNCTION_BLOCK Node_F_VN_ReadBarcodeExp2 EXTENDS VisionNode
VAR
    ipSrcImage : _ITcVnImage;
    ipDecodedData : _ITcVnContainer;
	ipContours : _ITcVnContainer;
    eBarcodeType : _ETcVnBarcodeType(ETcVnBarcodeType.TCVN_BT_ANY);
	nCodeNumber : _DINT(1);
	eSearchDirection : _ETcVnBarcodeSearchDirection(ETcVnBarcodeSearchDirection.TCVN_BSD_ANY);
	ipAngles : _ITcVnContainer; 
    hrPrev : _HRESULT(S_OK);
	hresult : _HRESULT(S_OK);
END_VAR

METHOD FB_init : BOOL
VAR_INPUT
	bInitRetains : BOOL; // if TRUE, the retain variables are initialized (warm start / cold start)
	bInCopyCode : BOOL;  // if TRUE, the instance afterwards gets moved into the copy code (online change)
END_VAR
AddInput('ipSrcImage', ipSrcImage);
AddParameter('eBarcodeType', eBarcodeType);
AddParameter('nCodeNumber', nCodeNumber);
AddParameter('eSearchDirection', eSearchDirection);
AddInput('hrPrev', hrPrev);
AddOutput('ipDecodedData', ipDecodedData);
AddOutput('ipContours', ipContours);
AddOutput('ipAngles', ipAngles);
AddOutput('hresult',hresult);
END_METHOD

METHOD PUBLIC  Clone : I_Node
VAR
	pNode : POINTER TO Node_F_VN_ReadBarcodeExp2;
END_VAR
pNode := __NEW(Node_F_VN_ReadBarcodeExp2);
Clone := pNode^;
END_METHOD

METHOD PROTECTED OnExecute
hresult.Value := F_VN_ReadBarcodeExp2(
	ipSrcImage := ipSrcImage.Value,
    ipDecodedData := ipDecodedData.Value,
	ipContours := ipContours.Value,
    eBarcodeType := eBarcodeType.Value,
	nCodeNumber := nCodeNumber.Value,
	eSearchDirection := eSearchDirection.Value,
	ipAngles := ipAngles.Value,
	hrPrev:= hrPrev.Value);
END_METHOD

METHOD PUBLIC PreExecutionCheck
VAR_INPUT
	Check : I_PreExecutionChecks;
END_VAR
Check.IsTrue(ipSrcImage.IsValid, 'ipSrcImage must contain an image');
Check.IsTrue((ipSrcImage.HasChannelCount(1) OR ipSrcImage.HasChannelCount(3)), 'ipSrcImage must have 1 or 3 channels');
Check.IsTrue(ipSrcImage.IsPixelDepth(8), 'ipSrcImage must have 8 bit pixel depth');
Check.IsTrue((nCodeNumber.Value = 1), 'nCodeNumber, currently only 1 supported');
END_METHOD

END_FUNCTION_BLOCK

// Nodes/Code Reading/Node_F_VN_ReadBarcodeRoi
{attribute 'linkalways'}
{attribute 'no_explicit_call' := 'This FB is a CLASS and must be accessed using methods or properties'}
{attribute 'enable_dynamic_creation'}
FUNCTION_BLOCK Node_F_VN_ReadBarcodeRoi EXTENDS VisionNode
VAR
    ipSrcImage : _ITcVnImage;
    ipDecodedData : _ITcVnContainer;
    eBarcodeType : _ETcVnBarcodeType(ETcVnBarcodeType.TCVN_BT_CODE128);
    hrPrev : _HRESULT(S_OK);
    fAngleDeg : _REAL(0);
    hresult : _HRESULT(S_OK);
END_VAR

METHOD FB_init : BOOL
VAR_INPUT
    bInitRetains : BOOL;
    bInCopyCode : BOOL;
END_VAR
AddInput('ipSrcImage', ipSrcImage);
AddOutput('ipDecodedData', ipDecodedData);
AddParameter('eBarcodeType', eBarcodeType);
AddInput('hrPrev', hrPrev);
AddOutput('fAngleDeg', fAngleDeg);
AddOutput('hresult', hresult);
END_METHOD

METHOD PUBLIC Clone : I_Node
VAR
    pNode : POINTER TO Node_F_VN_ReadBarcodeRoi;
END_VAR
pNode := __NEW(Node_F_VN_ReadBarcodeRoi);
Clone := pNode^;
END_METHOD

METHOD PROTECTED OnExecute
VAR
    angleDeg : REAL;
END_VAR
hresult.Value := F_VN_ReadBarcodeRoi(
    ipSrcImage := ipSrcImage.Value,
    ipDecodedData := ipDecodedData.Value,
    eBarcodeType := eBarcodeType.Value,
    hrPrev := hrPrev.Value,
    fAngleDeg => angleDeg);

fAngleDeg.Value := angleDeg;
END_METHOD

METHOD PUBLIC PreExecutionCheck
VAR_INPUT
    Check : I_PreExecutionChecks;
END_VAR
Check.IsTrue(ipSrcImage.IsValid, 'ipSrcImage must contain an image');
Check.IsTrue(ipSrcImage.HasChannelCount(1), 'ipSrcImage must contain 1 channel');
Check.IsTrue(ipSrcImage.IsPixelDepth(8), 'ipSrcImage must have 8 bit pixel depth');
Check.IsTrue((eBarcodeType.Value = ETcVnBarcodeType.TCVN_BT_CODE39) OR
             (eBarcodeType.Value = ETcVnBarcodeType.TCVN_BT_CODE128) OR
             (eBarcodeType.Value = ETcVnBarcodeType.TCVN_BT_EAN8) OR
             (eBarcodeType.Value = ETcVnBarcodeType.TCVN_BT_EAN13) OR
             (eBarcodeType.Value = ETcVnBarcodeType.TCVN_BT_ITF) OR
             (eBarcodeType.Value = ETcVnBarcodeType.TCVN_BT_UPCA) OR
             (eBarcodeType.Value = ETcVnBarcodeType.TCVN_BT_UPCE), 'eBarcodeType must be one of CODE39, CODE128, EAN8, EAN13, ITF, UPCA or UPCE');
END_METHOD

END_FUNCTION_BLOCK

// Nodes/Code Reading/Node_F_VN_ReadBarcodeRoiExp
{attribute 'linkalways'}
{attribute 'no_explicit_call' := 'This FB is a CLASS and must be accessed using methods or properties'}
{attribute 'enable_dynamic_creation'}
FUNCTION_BLOCK Node_F_VN_ReadBarcodeRoiExp EXTENDS VisionNode
VAR
    ipSrcImage : _ITcVnImage;
    ipDecodedData : _ITcVnContainer;
    eBarcodeType : _ETcVnBarcodeType(ETcVnBarcodeType.TCVN_BT_CODE128);
    eSearchDirection : _ETcVnBarcodeSearchDirection(ETcVnBarcodeSearchDirection.TCVN_BSD_ANY);
    ipContour : _ITcVnContainer;
    nMaxScans : _DINT(30);
    hrPrev : _HRESULT(S_OK);
    fAngleDeg : _REAL(0);
    hresult : _HRESULT(S_OK);
END_VAR

METHOD FB_init : BOOL
VAR_INPUT
    bInitRetains : BOOL;
    bInCopyCode : BOOL;
END_VAR
AddInput('ipSrcImage', ipSrcImage);
AddOutput('ipDecodedData', ipDecodedData);
AddParameter('eBarcodeType', eBarcodeType);
AddParameter('eSearchDirection', eSearchDirection);
AddOutput('ipContour', ipContour);
AddParameter('nMaxScans', nMaxScans);
AddInput('hrPrev', hrPrev);
AddOutput('fAngleDeg', fAngleDeg);
AddOutput('hresult', hresult);
END_METHOD

METHOD PUBLIC Clone : I_Node
VAR
    pNode : POINTER TO Node_F_VN_ReadBarcodeRoiExp;
END_VAR
pNode := __NEW(Node_F_VN_ReadBarcodeRoiExp);
Clone := pNode^;
END_METHOD

METHOD PROTECTED OnExecute
VAR
    angleDeg : REAL;
END_VAR
hresult.Value := F_VN_ReadBarcodeRoiExp(
    ipSrcImage := ipSrcImage.Value,
    ipDecodedData := ipDecodedData.Value,
    eBarcodeType := eBarcodeType.Value,
    eSearchDirection := eSearchDirection.Value,
    ipContour := ipContour.Value,
    nMaxScans := nMaxScans.Value,
    hrPrev := hrPrev.Value,
    fAngleDeg => angleDeg);

fAngleDeg.Value := angleDeg;
END_METHOD

METHOD PUBLIC PreExecutionCheck
VAR_INPUT
    Check : I_PreExecutionChecks;
END_VAR
Check.IsTrue(ipSrcImage.IsValid, 'ipSrcImage must contain an image');
Check.IsTrue(ipSrcImage.HasChannelCount(1), 'ipSrcImage must contain 1 channel');
Check.IsTrue(ipSrcImage.IsPixelDepth(8), 'ipSrcImage must have 8 bit pixel depth');
Check.IsTrue((eBarcodeType.Value = ETcVnBarcodeType.TCVN_BT_CODE39) OR
             (eBarcodeType.Value = ETcVnBarcodeType.TCVN_BT_CODE128) OR
             (eBarcodeType.Value = ETcVnBarcodeType.TCVN_BT_EAN8) OR
             (eBarcodeType.Value = ETcVnBarcodeType.TCVN_BT_EAN13) OR
             (eBarcodeType.Value = ETcVnBarcodeType.TCVN_BT_ITF) OR
             (eBarcodeType.Value = ETcVnBarcodeType.TCVN_BT_UPCA) OR
             (eBarcodeType.Value = ETcVnBarcodeType.TCVN_BT_UPCE), 'eBarcodeType must be one of CODE39, CODE128, EAN8, EAN13, ITF, UPCA or UPCE');
Check.IsTrue((eSearchDirection.Value = ETcVnBarcodeSearchDirection.TCVN_BSD_ANY) OR
             (eSearchDirection.Value = ETcVnBarcodeSearchDirection.TCVN_BSD_HORIZONTAL) OR
             (eSearchDirection.Value = ETcVnBarcodeSearchDirection.TCVN_BSD_VERTICAL), 'Unsupported eSearchDirection');
Check.IsTrue(nMaxScans.Value > 0, 'nMaxScans must be greater than 0');
END_METHOD

END_FUNCTION_BLOCK

// Nodes/Code Reading/Node_F_VN_ReadDataMatrixCode
{attribute 'linkalways'} 
{attribute 'no_explicit_call' := 'This FB is a CLASS and must be accessed using methods or properties'}
{attribute 'enable_dynamic_creation'}
FUNCTION_BLOCK Node_F_VN_ReadDataMatrixCode EXTENDS VisionNode
VAR
    ipSrcImage : _ITcVnImage;
    ipDecodedData : _ITcVnContainer;
    hrPrev : _HRESULT(S_OK);
	hresult : _HRESULT(S_OK);
END_VAR

METHOD FB_init : BOOL
VAR_INPUT
	bInitRetains : BOOL; // if TRUE, the retain variables are initialized (warm start / cold start)
	bInCopyCode : BOOL;  // if TRUE, the instance afterwards gets moved into the copy code (online change)
END_VAR
AddInput('ipSrcImage', ipSrcImage);
AddInput('hrPrev', hrPrev);
AddOutput('ipDecodedData', ipDecodedData);
AddOutput('hresult',hresult);
END_METHOD

METHOD PUBLIC  Clone : I_Node
VAR
	pNode : POINTER TO Node_F_VN_ReadDataMatrixCode;
END_VAR
pNode := __NEW(Node_F_VN_ReadDataMatrixCode);
Clone := pNode^;
END_METHOD

METHOD PROTECTED OnExecute
hresult.Value := F_VN_ReadDataMatrixCode(
	ipSrcImage := ipSrcImage.Value,
    ipDecodedData := ipDecodedData.Value,
	hrPrev:= hrPrev.Value);
END_METHOD

METHOD PUBLIC PreExecutionCheck
VAR_INPUT
	Check : I_PreExecutionChecks;
END_VAR
Check.IsTrue(ipSrcImage.IsValid, 'ipSrcImage must contain an image');
Check.IsTrue((ipSrcImage.HasChannelCount(1) OR ipSrcImage.HasChannelCount(3)), 'ipSrcImage must have 1 or 3 channels');
Check.IsTrue(ipSrcImage.IsPixelDepth(8), 'ipSrcImage must have 8 bit pixel depth');
END_METHOD

END_FUNCTION_BLOCK

// Nodes/Code Reading/Node_F_VN_ReadDataMatrixCodeExp
{attribute 'linkalways'} 
{attribute 'no_explicit_call' := 'This FB is a CLASS and must be accessed using methods or properties'}
{attribute 'enable_dynamic_creation'}
FUNCTION_BLOCK Node_F_VN_ReadDataMatrixCodeExp EXTENDS VisionNode
VAR
    ipSrcImage : _ITcVnImage;
    ipDecodedData : _ITcVnContainer;
	ipContours : _ITcVnContainer;
	nCodeNumber : _DINT(1);
	eSearchStrategy : _UDINT(ETcVn2dCodeSearchStrategy.TCVN_CSS_DEFAULT);
    hrPrev : _HRESULT(S_OK);
	hresult : _HRESULT(S_OK);
END_VAR

METHOD FB_init : BOOL
VAR_INPUT
	bInitRetains : BOOL; // if TRUE, the retain variables are initialized (warm start / cold start)
	bInCopyCode : BOOL;  // if TRUE, the instance afterwards gets moved into the copy code (online change)
END_VAR
AddInput('ipSrcImage', ipSrcImage);
AddInput('hrPrev', hrPrev);
AddParameter('nCodeNumber',nCodeNumber);
AddParameter('eSearchStrategy',eSearchStrategy);
AddOutput('ipDecodedData', ipDecodedData);
AddOutput('ipContours', ipContours);
AddOutput('hresult',hresult);
END_METHOD

METHOD PUBLIC  Clone : I_Node
VAR
	pNode : POINTER TO Node_F_VN_ReadDataMatrixCodeExp;
END_VAR
pNode := __NEW(Node_F_VN_ReadDataMatrixCodeExp);
Clone := pNode^;
END_METHOD

METHOD PROTECTED OnExecute
hresult.Value := F_VN_ReadDataMatrixCodeExp(
	ipSrcImage := ipSrcImage.Value,
    ipDecodedData := ipDecodedData.Value,
	ipContours := ipContours.Value,
	nCodeNumber := nCodeNumber.Value,
	eSearchStrategy := eSearchStrategy.Value,	
	hrPrev:= hrPrev.Value);
END_METHOD

METHOD PUBLIC PreExecutionCheck
VAR_INPUT
	Check : I_PreExecutionChecks;
END_VAR
Check.IsTrue(ipSrcImage.IsValid, 'ipSrcImage must contain an image');
Check.IsTrue((ipSrcImage.HasChannelCount(1) OR ipSrcImage.HasChannelCount(3)), 'ipSrcImage must have 1 or 3 channels');
Check.IsTrue(ipSrcImage.IsPixelDepth(8), 'ipSrcImage must have 8 bit pixel depth');
Check.IsTrue((nCodeNumber.Value = 1), 'nCodeNumber, currently only 1 supported');
END_METHOD

END_FUNCTION_BLOCK

// Nodes/Code Reading/Node_F_VN_ReadDataMatrixCodeExp2
{attribute 'linkalways'} 
{attribute 'no_explicit_call' := 'This FB is a CLASS and must be accessed using methods or properties'}
{attribute 'enable_dynamic_creation'}
FUNCTION_BLOCK Node_F_VN_ReadDataMatrixCodeExp2 EXTENDS VisionNode
VAR
    ipSrcImage : _ITcVnImage;
    ipDecodedData : _ITcVnContainer;
	ipContours : _ITcVnContainer;
	nCodeNumber : _DINT(1);
	eSearchStrategy : _UDINT(ETcVn2dCodeSearchStrategy.TCVN_CSS_DEFAULT);
	ipAngles : _ITcVnContainer;
    hrPrev : _HRESULT(S_OK);
	hresult : _HRESULT(S_OK);
END_VAR

METHOD FB_init : BOOL
VAR_INPUT
	bInitRetains : BOOL; // if TRUE, the retain variables are initialized (warm start / cold start)
	bInCopyCode : BOOL;  // if TRUE, the instance afterwards gets moved into the copy code (online change)
END_VAR
AddInput('ipSrcImage', ipSrcImage);
AddInput('hrPrev', hrPrev);
AddParameter('nCodeNumber',nCodeNumber);
AddParameter('eSearchStrategy',eSearchStrategy);
AddOutput('ipDecodedData', ipDecodedData);
AddOutput('ipContours', ipContours);
AddOutput('ipAngles', ipAngles);
AddOutput('hresult',hresult);
END_METHOD

METHOD PUBLIC  Clone : I_Node
VAR
	pNode : POINTER TO Node_F_VN_ReadDataMatrixCodeExp2;
END_VAR
pNode := __NEW(Node_F_VN_ReadDataMatrixCodeExp2);
Clone := pNode^;
END_METHOD

METHOD PROTECTED OnExecute
hresult.Value := F_VN_ReadDataMatrixCodeExp2(
	ipSrcImage := ipSrcImage.Value,
    ipDecodedData := ipDecodedData.Value,
	ipContours := ipContours.Value,
	nCodeNumber := nCodeNumber.Value,
	eSearchStrategy := eSearchStrategy.Value,
	ipAngles := ipAngles.Value,
	hrPrev:= hrPrev.Value);
END_METHOD

METHOD PUBLIC PreExecutionCheck
VAR_INPUT
	Check : I_PreExecutionChecks;
END_VAR
Check.IsTrue(ipSrcImage.IsValid, 'ipSrcImage must contain an image');
Check.IsTrue((ipSrcImage.HasChannelCount(1) OR ipSrcImage.HasChannelCount(3)), 'ipSrcImage must have 1 or 3 channels');
Check.IsTrue(ipSrcImage.IsPixelDepth(8), 'ipSrcImage must have 8 bit pixel depth');
Check.IsTrue((nCodeNumber.Value = 1), 'nCodeNumber, currently only 1 supported');
END_METHOD

END_FUNCTION_BLOCK

// Nodes/Code Reading/Node_F_VN_ReadDataMatrixCodeRoi
{attribute 'linkalways'} 
{attribute 'no_explicit_call' := 'This FB is a CLASS and must be accessed using methods or properties'}
{attribute 'enable_dynamic_creation'}
FUNCTION_BLOCK Node_F_VN_ReadDataMatrixCodeRoi EXTENDS VisionNode
VAR
    ipSrcImage : _ITcVnImage;
    ipDecodedData : _ITcVnContainer;
    fModuleWidth : _REAL(3);
    hrPrev : _HRESULT(S_OK);
	fAngleDeg : _REAL(0);
	hresult : _HRESULT(S_OK);
END_VAR

METHOD FB_init : BOOL
VAR_INPUT
	bInitRetains : BOOL; // if TRUE, the retain variables are initialized (warm start / cold start)
	bInCopyCode : BOOL;  // if TRUE, the instance afterwards gets moved into the copy code (online change)
END_VAR
AddInput('ipSrcImage', ipSrcImage);
AddOutput('ipDecodedData', ipDecodedData);
AddParameter('fModuleWidth', fModuleWidth);
AddInput('hrPrev', hrPrev);
AddOutput('fAngleDeg', fAngleDeg);
AddOutput('hresult', hresult);
END_METHOD

METHOD PUBLIC  Clone : I_Node
VAR
	pNode : POINTER TO Node_F_VN_ReadDataMatrixCodeRoi;
END_VAR
pNode := __NEW(Node_F_VN_ReadDataMatrixCodeRoi);
Clone := pNode^;
END_METHOD

METHOD PROTECTED OnExecute
VAR
	tempfAngleDeg : REAL;
END_VAR
hresult.Value := F_VN_ReadDataMatrixCodeRoi(
	ipSrcImage := ipSrcImage.Value,
    ipDecodedData := ipDecodedData.Value,
    fModuleWidth := fModuleWidth.Value,
	hrPrev:= hrPrev.Value,
	fAngleDeg => tempfAngleDeg
);

IF succeeded(hresult.Value) THEN
	fAngleDeg.Value := tempfAngleDeg;
END_IF
END_METHOD

METHOD PUBLIC PreExecutionCheck
VAR_INPUT
	Check : I_PreExecutionChecks;
END_VAR
Check.IsTrue(ipSrcImage.IsValid, 'ipSrcImage must contain an image');
Check.IsTrue((ipSrcImage.IsPixelDepth(8)), 'ipSrcImage must be 8 bit pixel depth');
Check.IsTrue((ipSrcImage.HasChannelCount(1)), 'ipSrcImage must contain 1 channel');
Check.IsTrue((fModuleWidth.Value >= 3), 'fModuleWidth must be at least 3, preferably 5 - 8.');
END_METHOD

END_FUNCTION_BLOCK

// Nodes/Code Reading/Node_F_VN_ReadDataMatrixCodeRoiExp
{attribute 'linkalways'}
{attribute 'no_explicit_call' := 'This FB is a CLASS and must be accessed using methods or properties'}
{attribute 'enable_dynamic_creation'}
FUNCTION_BLOCK Node_F_VN_ReadDataMatrixCodeRoiExp EXTENDS VisionNode
VAR
    ipSrcImage : _ITcVnImage;
    ipDecodedData : _ITcVnContainer;
    fModuleWidth : _REAL(3);
    ipContour : _ITcVnContainer;
    eOptions : _ULINT(ETcVnDataMatrixOptions.TCVN_DMO_DEFAULT);
    nRows : _USINT(0);
    nCols : _USINT(0);
    bExtensiveSearch : _BOOL(TRUE);
    hrPrev : _HRESULT(S_OK);
    fAngleDeg : _REAL(0);
    hresult : _HRESULT(S_OK);
END_VAR

METHOD FB_init : BOOL
VAR_INPUT
    bInitRetains : BOOL;
    bInCopyCode : BOOL;
END_VAR
AddInput('ipSrcImage', ipSrcImage);
AddOutput('ipDecodedData', ipDecodedData);
AddParameter('fModuleWidth', fModuleWidth);
AddOutput('ipContour', ipContour);
AddParameter('eOptions', eOptions);
AddParameter('nRows', nRows);
AddParameter('nCols', nCols);
AddParameter('bExtensiveSearch', bExtensiveSearch);
AddInput('hrPrev', hrPrev);
AddOutput('fAngleDeg', fAngleDeg);
AddOutput('hresult', hresult);
END_METHOD

METHOD PUBLIC Clone : I_Node
VAR
    pNode : POINTER TO Node_F_VN_ReadDataMatrixCodeRoiExp;
END_VAR
pNode := __NEW(Node_F_VN_ReadDataMatrixCodeRoiExp);
Clone := pNode^;
END_METHOD

METHOD PROTECTED OnExecute
VAR
    angleDeg : REAL;
END_VAR
hresult.Value := F_VN_ReadDataMatrixCodeRoiExp(
    ipSrcImage := ipSrcImage.Value,
    ipDecodedData := ipDecodedData.Value,
    fModuleWidth := fModuleWidth.Value,
    ipContour := ipContour.Value,
    eOptions := eOptions.Value,
    nRows := nRows.Value,
    nCols := nCols.Value,
    bExtensiveSearch := bExtensiveSearch.Value,
    hrPrev := hrPrev.Value,
    fAngleDeg => angleDeg);

fAngleDeg.Value := angleDeg;
END_METHOD

METHOD PUBLIC PreExecutionCheck
VAR_INPUT
    Check : I_PreExecutionChecks;
END_VAR
Check.IsTrue(ipSrcImage.IsValid, 'ipSrcImage must contain an image');
Check.IsTrue(ipSrcImage.HasChannelCount(1), 'ipSrcImage must contain 1 channel');
Check.IsTrue(ipSrcImage.IsPixelDepth(8), 'ipSrcImage must have 8 bit pixel depth');
Check.IsTrue(fModuleWidth.Value >= 3.0, 'fModuleWidth must be at least 3');
// 0 searches for any size.
Check.IsTrue((nRows.Value = 0) OR ((nRows.Value >= 8) AND (nRows.Value <= 144)), 'nRows must be 0 to search any size, or between 8 and 144');
Check.IsTrue((nCols.Value = 0) OR ((nCols.Value >= 10) AND (nCols.Value <= 144)), 'nCols must be 0 to search any size, or between 10 and 144');
END_METHOD

END_FUNCTION_BLOCK

// Nodes/Code Reading/Node_F_VN_ReadDotCodeRoi
{attribute 'linkalways'} 
{attribute 'no_explicit_call' := 'This FB is a CLASS and must be accessed using methods or properties'}
{attribute 'enable_dynamic_creation'}
FUNCTION_BLOCK Node_F_VN_ReadDotCodeRoi EXTENDS VisionNode
VAR
    ipSrcImage : _ITcVnImage;
    ipDecodedData : _ITcVnContainer;
	fModuleWidth : _REAL(3);
    hrPrev : _HRESULT(S_OK);
	fAngleDeg : _REAL(0);
	hresult : _HRESULT(S_OK);
END_VAR

METHOD FB_init : BOOL
VAR_INPUT
	bInitRetains : BOOL; // if TRUE, the retain variables are initialized (warm start / cold start)
	bInCopyCode : BOOL;  // if TRUE, the instance afterwards gets moved into the copy code (online change)
END_VAR
AddInput('ipSrcImage', ipSrcImage);
AddInput('fModuleWidth', fModuleWidth);
AddInput('hrPrev', hrPrev);
AddOutput('ipDecodedData', ipDecodedData);
AddOutput('fAngleDeg',fAngleDeg);
AddOutput('hresult',hresult);
END_METHOD

METHOD PUBLIC  Clone : I_Node
VAR
	pNode : POINTER TO Node_F_VN_ReadDotCodeRoi;
END_VAR
pNode := __NEW(Node_F_VN_ReadDotCodeRoi);
Clone := pNode^;
END_METHOD

METHOD PROTECTED OnExecute
VAR
	_fAngleDeg : REAL;
END_VAR
hresult.Value := F_VN_ReadDotCodeRoi(
	ipSrcImage := ipSrcImage.Value,
    ipDecodedData := ipDecodedData.Value,
	fModuleWidth := fModuleWidth.Value,
	hrPrev:= hrPrev.Value,
	fAngleDeg => _fAngleDeg);
	
fAngleDeg.Value := _fAngleDeg;
END_METHOD

METHOD PUBLIC PreExecutionCheck
VAR_INPUT
	Check : I_PreExecutionChecks;
END_VAR
Check.IsTrue(ipSrcImage.IsValid, 'ipSrcImage must contain an image');
Check.IsTrue(ipSrcImage.HasChannelCount(1), 'ipSrcImage must have 1 channels');
Check.IsTrue(fModuleWidth.Value >= 3, 'fModuleWidth must be equal or greter than 3 (preferably 5 - 8)');
Check.IsTrue(ipSrcImage.IsElementType(ETcVnElementType.TCVN_ET_USINT), 'ipSrcImage must have an element type of USINT');
END_METHOD

END_FUNCTION_BLOCK

// Nodes/Code Reading/Node_F_VN_ReadDotCodeRoiExp
{attribute 'linkalways'} 
{attribute 'no_explicit_call' := 'This FB is a CLASS and must be accessed using methods or properties'}
{attribute 'enable_dynamic_creation'}
FUNCTION_BLOCK Node_F_VN_ReadDotCodeRoiExp EXTENDS VisionNode
VAR
    ipSrcImage : _ITcVnImage;
    ipDecodedData : _ITcVnContainer;
	fModuleWidth : _REAL(3);
	eOptions : _ULINT(ETcVnDotCodeOptions.TCVN_DCO_DEFAULT);
	ipContour : _ITcVnContainer;
    hrPrev : _HRESULT(S_OK);
	fAngleDeg : _REAL(0);
	hresult : _HRESULT(S_OK);
END_VAR

METHOD FB_init : BOOL
VAR_INPUT
	bInitRetains : BOOL; // if TRUE, the retain variables are initialized (warm start / cold start)
	bInCopyCode : BOOL;  // if TRUE, the instance afterwards gets moved into the copy code (online change)
END_VAR
AddInput('ipSrcImage', ipSrcImage);
AddInput('fModuleWidth', fModuleWidth);
AddInput('eOptions', eOptions);
AddInput('hrPrev', hrPrev);
AddOutput('ipDecodedData', ipDecodedData);
AddOutput('ipContour', ipContour);
AddOutput('fAngleDeg',fAngleDeg);
AddOutput('hresult',hresult);
END_METHOD

METHOD PUBLIC  Clone : I_Node
VAR
	pNode : POINTER TO Node_F_VN_ReadDotCodeRoiExp;
END_VAR
pNode := __NEW(Node_F_VN_ReadDotCodeRoiExp);
Clone := pNode^;
END_METHOD

METHOD PROTECTED OnExecute
VAR
	_fAngleDeg : REAL;
END_VAR
hresult.Value := F_VN_ReadDotCodeRoiExp(
	ipSrcImage := ipSrcImage.Value,
    ipDecodedData := ipDecodedData.Value,
	fModuleWidth := fModuleWidth.Value,
	ipContour := ipContour.Value,
	eOptions := eOptions.Value,
	hrPrev:= hrPrev.Value,
	fAngleDeg => _fAngleDeg);
	
fAngleDeg.Value := _fAngleDeg;
END_METHOD

METHOD PUBLIC PreExecutionCheck
VAR_INPUT
	Check : I_PreExecutionChecks;
END_VAR
Check.IsTrue(ipSrcImage.IsValid, 'ipSrcImage must contain an image');
Check.IsTrue(ipSrcImage.HasChannelCount(1), 'ipSrcImage must have 1 channels');
Check.IsTrue(fModuleWidth.Value >= 3, 'fModuleWidth must be equal or greter than 3 (preferably 5 - 8)');
Check.IsTrue(ipSrcImage.IsElementType(ETcVnElementType.TCVN_ET_USINT), 'ipSrcImage must have an element type of USINT');
END_METHOD

END_FUNCTION_BLOCK

// Nodes/Code Reading/Node_F_VN_ReadPharmaCode
{attribute 'linkalways'} 
{attribute 'no_explicit_call' := 'This FB is a CLASS and must be accessed using methods or properties'}
{attribute 'enable_dynamic_creation'}
FUNCTION_BLOCK Node_F_VN_ReadPharmaCode EXTENDS VisionNode
VAR
    ipSrcImage : _ITcVnImage;
    ipDecodedData : _ITcVnContainer;
    hrPrev : _HRESULT(S_OK);
	hresult : _HRESULT(S_OK);
END_VAR

METHOD FB_init : BOOL
VAR_INPUT
	bInitRetains : BOOL; // if TRUE, the retain variables are initialized (warm start / cold start)
	bInCopyCode : BOOL;  // if TRUE, the instance afterwards gets moved into the copy code (online change)
END_VAR
AddInput('ipSrcImage', ipSrcImage);
AddInput('hrPrev', hrPrev);
AddOutput('ipDecodedData', ipDecodedData);
AddOutput('hresult',hresult);
END_METHOD

METHOD PUBLIC  Clone : I_Node
VAR
	pNode : POINTER TO Node_F_VN_ReadPharmaCode;
END_VAR
pNode := __NEW(Node_F_VN_ReadPharmaCode);
Clone := pNode^;
END_METHOD

METHOD PROTECTED OnExecute
hresult.Value := F_VN_ReadPharmaCode(
	ipSrcImage := ipSrcImage.Value,
    ipDecodedData := ipDecodedData.Value,
	hrPrev:= hrPrev.Value);
END_METHOD

METHOD PUBLIC PreExecutionCheck
VAR_INPUT
	Check : I_PreExecutionChecks;
END_VAR
Check.IsTrue(ipSrcImage.IsValid, 'ipSrcImage must contain an image');
Check.IsTrue((ipSrcImage.HasChannelCount(1) OR ipSrcImage.HasChannelCount(3)), 'ipSrcImage must have 1 or 3 channels');

IF (ipSrcImage.HasChannelCount(1)) THEN
    Check.IsTrue(ipSrcImage.IsPixelDepth(8), 'ipSrcImage must have 8 bit pixel depth');
END_IF

IF (ipSrcImage.HasChannelCount(3)) THEN
    Check.IsTrue((ipSrcImage.IsPixelDepth(8) OR 
                 ipSrcImage.IsPixelDepth(16) OR
                 ipSrcImage.IsPixelDepth(32)), 'ipSrcImage must have 8, 16 or 32 bit pixel depth');
END_IF
END_METHOD

END_FUNCTION_BLOCK

// Nodes/Code Reading/Node_F_VN_ReadPharmaCodeExp
{attribute 'linkalways'} 
{attribute 'no_explicit_call' := 'This FB is a CLASS and must be accessed using methods or properties'}
{attribute 'enable_dynamic_creation'}
FUNCTION_BLOCK Node_F_VN_ReadPharmaCodeExp EXTENDS VisionNode
VAR
    ipSrcImage : _ITcVnImage;
    ipDecodedData : _ITcVnContainer;
	ipContours : _ITcVnContainer;
	nCodeNumber : _DINT(1);
	nMinBarNumber : _INT(4);
    hrPrev : _HRESULT(S_OK);
	hresult : _HRESULT(S_OK);
END_VAR

METHOD FB_init : BOOL
VAR_INPUT
	bInitRetains : BOOL; // if TRUE, the retain variables are initialized (warm start / cold start)
	bInCopyCode : BOOL;  // if TRUE, the instance afterwards gets moved into the copy code (online change)
END_VAR
AddInput('ipSrcImage', ipSrcImage);
AddInput('hrPrev', hrPrev);
AddParameter('nCodeNumber',nCodeNumber);
AddParameter('nMinBarNumber',nMinBarNumber);
AddOutput('ipDecodedData', ipDecodedData);
AddOutput('ipContours', ipDecodedData);
AddOutput('hresult',hresult);
END_METHOD

METHOD PUBLIC  Clone : I_Node
VAR
	pNode : POINTER TO Node_F_VN_ReadPharmaCodeExp;
END_VAR
pNode := __NEW(Node_F_VN_ReadPharmaCodeExp);
Clone := pNode^;
END_METHOD

METHOD PROTECTED OnExecute
hresult.Value := F_VN_ReadPharmaCodeExp(
	ipSrcImage := ipSrcImage.Value,
    ipDecodedData := ipDecodedData.Value,
	ipContours := ipContours.Value,
	nCodeNumber := nCodeNumber.Value,
	nMinBarNumber := nMinBarNumber.Value,
	hrPrev:= hrPrev.Value);
END_METHOD

METHOD PUBLIC PreExecutionCheck
VAR_INPUT
	Check : I_PreExecutionChecks;
END_VAR
Check.IsTrue(ipSrcImage.IsValid, 'ipSrcImage must contain an image');
Check.IsTrue((ipSrcImage.HasChannelCount(1) OR ipSrcImage.HasChannelCount(3)), 'ipSrcImage must have 1 or 3 channels');

IF (ipSrcImage.HasChannelCount(1)) THEN
    Check.IsTrue(ipSrcImage.IsPixelDepth(8), 'ipSrcImage must have 8 bit pixel depth');
END_IF

IF (ipSrcImage.HasChannelCount(3)) THEN
    Check.IsTrue((ipSrcImage.IsPixelDepth(8) OR 
                 ipSrcImage.IsPixelDepth(16) OR
                 ipSrcImage.IsPixelDepth(32)), 'ipSrcImage must have 8, 16 or 32 bit pixel depth');
END_IF

Check.IsTrue((nCodeNumber.Value = 1), 'nCodeNumber, currently only 1 supported');
END_METHOD

END_FUNCTION_BLOCK

